LIN {X 0,Y 516.86,Z 224.104,A -85,B 0,C 180,E1 -4913.251,E2 -4913.251} C_VEL
LIN {X 0,Y 516.891,Z 224.097,A -85,B 0,C 180,E1 -4916.118,E2 -4916.118} C_VEL
LIN {X 0,Y 516.796,Z 224.113,A -85,B 0,C 180,E1 -4918.954,E2 -4918.954} C_VEL
LIN {X 0,Y 516.6,Z 224.138,A -85,B 0,C 180,E1 -4920.674,E2 -4920.674} C_VEL
LIN {X 0,Y 516.555,Z 225.784,A -85,B 0,C 180,E1 -4922.445,E2 -4922.445} C_VEL
LIN {X 0,Y 516.513,Z 229.358,A -85,B 0,C 180,E1 -4925.734,E2 -4925.734} C_VEL
LIN {X 0,Y 516.417,Z 232.326,A -85,B 0,C 180,E1 -4928.441,E2 -4928.441} C_VEL
LIN {X 0,Y 516.398,Z 235.073,A -85,B 0,C 180,E1 -4930.934,E2 -4930.934} C_VEL
LIN {X 0,Y 516.39,Z 237.798,A -85,B 0,C 180,E1 -4933.392,E2 -4933.392} C_VEL
LIN {X 0,Y 516.408,Z 240.566,A -85,B 0,C 180,E1 -4935.819,E2 -4935.819} C_VEL
LIN {X 0,Y 516.373,Z 244.264,A -85,B 0,C 180,E1 -4939.014,E2 -4939.014} C_VEL
LIN {X 0,Y 516.358,Z 245.702,A -85,B 0,C 180,E1 -4940.203,E2 -4940.203} C_VEL
LIN {X 0,Y 518.519,Z 256.334,A -85,B 0,C 180,E1 -4940.54,E2 -4940.54} C_VEL
LIN {X 0,Y 518.318,Z 269.35,A -85,B 0,C 180,E1 -4941.028,E2 -4941.028} C_VEL
LIN {X 0,Y 518.116,Z 280.838,A -85,B 0,C 180,E1 -4941.614,E2 -4941.614} C_VEL
LIN {X 0,Y 517.752,Z 291.503,A -85,B 0,C 180,E1 -4942.307,E2 -4942.307} C_VEL
LIN {X 0,Y 517.502,Z 302.062,A -85,B 0,C 180,E1 -4943.174,E2 -4943.174} C_VEL
LIN {X 0,Y 517.212,Z 311.692,A -85,B 0,C 180,E1 -4944.15,E2 -4944.15} C_VEL
LIN {X 0,Y 516.934,Z 319.598,A -85,B 0,C 180,E1 -4945.124,E2 -4945.124} C_VEL
LIN {X 0,Y 516.716,Z 327.363,A -85,B 0,C 180,E1 -4946.295,E2 -4946.295} C_VEL
LIN {X 0,Y 516.565,Z 332.623,A -85,B 0,C 180,E1 -4947.27,E2 -4947.27} C_VEL
LIN {X 0,Y 516.325,Z 337.788,A -85,B 0,C 180,E1 -4948.439,E2 -4948.439} C_VEL
LIN {X 0,Y 516.372,Z 341.79,A -85,B 0,C 180,E1 -4949.609,E2 -4949.609} C_VEL
LIN {X 0,Y 516.205,Z 344.784,A -85,B 0,C 180,E1 -4950.779,E2 -4950.779} C_VEL
LIN {X 0,Y 516.205,Z 346.261,A -85,B 0,C 180,E1 -4951.559,E2 -4951.559} C_VEL
LIN {X 0,Y 516.352,Z 347.941,A -85,B 0,C 180,E1 -4953.12,E2 -4953.12} C_VEL
LIN {X 0,Y 516.323,Z 348.221,A -85,B 0,C 180,E1 -4953.901,E2 -4953.901} C_VEL
LIN {X 0,Y 516.234,Z 348.118,A -85,B 0,C 180,E1 -4954.684,E2 -4954.684} C_VEL
LIN {X 0,Y 516.3,Z 347.579,A -85,B 0,C 180,E1 -4955.467,E2 -4955.467} C_VEL
LIN {X 0,Y 516.323,Z 345.343,A -85,B 0,C 180,E1 -4957.035,E2 -4957.035} C_VEL
LIN {X 0,Y 516.361,Z 342.554,A -85,B 0,C 180,E1 -4958.215,E2 -4958.215} C_VEL
LIN {X 0,Y 516.401,Z 338.739,A -85,B 0,C 180,E1 -4959.398,E2 -4959.398} C_VEL
LIN {X 0,Y 516.519,Z 333.78,A -85,B 0,C 180,E1 -4960.583,E2 -4960.583} C_VEL
LIN {X 0,Y 516.739,Z 327.523,A -85,B 0,C 180,E1 -4961.77,E2 -4961.77} C_VEL
LIN {X 0,Y 516.954,Z 319.645,A -85,B 0,C 180,E1 -4962.961,E2 -4962.961} C_VEL
LIN {X 0,Y 517.176,Z 311.578,A -85,B 0,C 180,E1 -4963.957,E2 -4963.957} C_VEL
LIN {X 0,Y 517.498,Z 301.699,A -85,B 0,C 180,E1 -4964.952,E2 -4964.952} C_VEL
LIN {X 0,Y 517.737,Z 291.95,A -85,B 0,C 180,E1 -4965.752,E2 -4965.752} C_VEL
LIN {X 0,Y 518.044,Z 281.356,A -85,B 0,C 180,E1 -4966.45,E2 -4966.45} C_VEL
LIN {X 0,Y 518.269,Z 268.518,A -85,B 0,C 180,E1 -4967.102,E2 -4967.102} C_VEL
LIN {X 0,Y 518.449,Z 255.755,A -85,B 0,C 180,E1 -4967.572,E2 -4967.572} C_VEL
LIN {X 0,Y 516.346,Z 245.639,A -85,B 0,C 180,E1 -4967.9,E2 -4967.9} C_VEL
LIN {X 0,Y 516.311,Z 242.393,A -85,B 0,C 180,E1 -4970.725,E2 -4970.725} C_VEL
LIN {X 0,Y 516.385,Z 239.494,A -85,B 0,C 180,E1 -4973.245,E2 -4973.245} C_VEL
LIN {X 0,Y 516.46,Z 236.317,A -85,B 0,C 180,E1 -4976.086,E2 -4976.086} C_VEL
LIN {X 0,Y 516.466,Z 233.733,A -85,B 0,C 180,E1 -4978.441,E2 -4978.441} C_VEL
LIN {X 0,Y 516.508,Z 230.848,A -85,B 0,C 180,E1 -4981.133,E2 -4981.133} C_VEL
LIN {X 0,Y 516.564,Z 227.881,A -85,B 0,C 180,E1 -4983.909,E2 -4983.909} C_VEL
LIN {X 0,Y 516.61,Z 224.866,A -85,B 0,C 180,E1 -4986.767,E2 -4986.767} C_VEL
LIN {X 0,Y 516.683,Z 224.128,A -85,B 0,C 180,E1 -4987.914,E2 -4987.914} C_VEL
LIN {X 0,Y 516.873,Z 224.101,A -85,B 0,C 180,E1 -4990.741,E2 -4990.741} C_VEL
LIN {X 0,Y 516.879,Z 224.103,A -85,B 0,C 180,E1 -4992.83,E2 -4992.83} C_VEL
LIN {X 0,Y 516.917,Z 224.094,A -85,B 0,C 180,E1 -4995.009,E2 -4995.009} C_VEL
LIN {X 0,Y 516.901,Z 224.096,A -85,B 0,C 180,E1 -4998.398,E2 -4998.398} C_VEL
LIN {X 0,Y 516.874,Z 224.101,A -85,B 0,C 180,E1 -5001.283,E2 -5001.283} C_VEL
LIN {X 0,Y 516.883,Z 224.103,A -85,B 0,C 180,E1 -5004.22,E2 -5004.22} C_VEL
LIN {X 0,Y 516.872,Z 224.1,A -85,B 0,C 180,E1 -5007.051,E2 -5007.051} C_VEL
LIN {X 0,Y 516.877,Z 224.099,A -85,B 0,C 180,E1 -5009.795,E2 -5009.795} C_VEL
LIN {X 0,Y 516.921,Z 224.097,A -85,B 0,C 180,E1 -5012.467,E2 -5012.467} C_VEL
LIN {X 0,Y 516.902,Z 224.095,A -85,B 0,C 180,E1 -5015.071,E2 -5015.071} C_VEL
LIN {X 0,Y 516.874,Z 224.099,A -85,B 0,C 180,E1 -5018.462,E2 -5018.462} C_VEL
LIN {X 0,Y 516.89,Z 224.1,A -85,B 0,C 180,E1 -5020.954,E2 -5020.954} C_VEL
LIN {X 0,Y 516.904,Z 224.096,A -85,B 0,C 180,E1 -5023.41,E2 -5023.41} C_VEL
LIN {X 0,Y 516.885,Z 224.101,A -85,B 0,C 180,E1 -5025.833,E2 -5025.833} C_VEL
LIN {X 0,Y 516.954,Z 224.089,A -85,B 0,C 180,E1 -5028.233,E2 -5028.233} C_VEL
LIN {X 0,Y 516.953,Z 224.089,A -85,B 0,C 180,E1 -5031.399,E2 -5031.399} C_VEL
LIN {X 0,Y 517.056,Z 224.077,A -85,B 0,C 180,E1 -5034.54,E2 -5034.54} C_VEL
LIN {X 0,Y 517.07,Z 224.075,A -85,B 0,C 180,E1 -5037.663,E2 -5037.663} C_VEL
LIN {X 0,Y 517.079,Z 224.076,A -85,B 0,C 180,E1 -5040.779,E2 -5040.779} C_VEL
LIN {X 0,Y 517.003,Z 224.083,A -85,B 0,C 180,E1 -5043.117,E2 -5043.117} C_VEL
LIN {X 0,Y 517.001,Z 224.083,A -85,B 0,C 180,E1 -5046.243,E2 -5046.243} C_VEL
LIN {X 0,Y 516.939,Z 224.091,A -85,B 0,C 180,E1 -5049.389,E2 -5049.389} C_VEL
LIN {X 0,Y 516.939,Z 224.094,A -85,B 0,C 180,E1 -5051.807,E2 -5051.807} C_VEL
LIN {X 0,Y 516.933,Z 224.095,A -85,B 0,C 180,E1 -5055.147,E2 -5055.147} C_VEL
LIN {X 0,Y 516.915,Z 224.095,A -85,B 0,C 180,E1 -5058.223,E2 -5058.223} C_VEL
LIN {X 0,Y 516.901,Z 224.097,A -85,B 0,C 180,E1 -5060.702,E2 -5060.702} C_VEL
LIN {X 0,Y 516.879,Z 224.099,A -85,B 0,C 180,E1 -5064.074,E2 -5064.074} C_VEL
LIN {X 0,Y 516.92,Z 224.097,A -85,B 0,C 180,E1 -5066.658,E2 -5066.658} C_VEL
LIN {X 0,Y 516.915,Z 224.094,A -85,B 0,C 180,E1 -5069.527,E2 -5069.527} C_VEL
LIN {X 0,Y 516.885,Z 224.098,A -85,B 0,C 180,E1 -5072.544,E2 -5072.544} C_VEL
LIN {X 0,Y 516.857,Z 224.104,A -85,B 0,C 180,E1 -5075.331,E2 -5075.331} C_VEL
LIN {X 0,Y 516.873,Z 224.1,A -85,B 0,C 180,E1 -5077.944,E2 -5077.944} C_VEL
LIN {X 0,Y 516.874,Z 224.099,A -85,B 0,C 180,E1 -5080.743,E2 -5080.743} C_VEL
LIN {X 0,Y 516.873,Z 224.1,A -85,B 0,C 180,E1 -5083.904,E2 -5083.904} C_VEL
LIN {X 0,Y 516.875,Z 224.102,A -85,B 0,C 180,E1 -5086.108,E2 -5086.108} C_VEL
LIN {X 0,Y 516.898,Z 224.1,A -85,B 0,C 180,E1 -5089.262,E2 -5089.262} C_VEL
LIN {X 0,Y 516.894,Z 224.132,A -85,B 0,C 180,E1 -5091.287,E2 -5091.287} C_VEL
LIN {X 0,Y 518.012,Z 230.689,A -85,B 0,C 180,E1 -5093.832,E2 -5093.832} C_VEL
LIN {X 0,Y 518.059,Z 236.321,A -85,B 0,C 180,E1 -5095.846,E2 -5095.846} C_VEL
LIN {X 0,Y 517.804,Z 244.803,A -85,B 0,C 180,E1 -5098.769,E2 -5098.769} C_VEL
LIN {X 0,Y 517.573,Z 254.623,A -85,B 0,C 180,E1 -5101.96,E2 -5101.96} C_VEL
LIN {X 0,Y 517.325,Z 262.962,A -85,B 0,C 180,E1 -5104.665,E2 -5104.665} C_VEL
LIN {X 0,Y 517.112,Z 272.229,A -85,B 0,C 180,E1 -5107.634,E2 -5107.634} C_VEL
LIN {X 0,Y 516.902,Z 281.496,A -85,B 0,C 180,E1 -5110.544,E2 -5110.544} C_VEL
LIN {X 0,Y 516.708,Z 290.764,A -85,B 0,C 180,E1 -5113.405,E2 -5113.405} C_VEL
LIN {X 0,Y 516.568,Z 299.534,A -85,B 0,C 180,E1 -5116.077,E2 -5116.077} C_VEL
LIN {X 0,Y 518.521,Z 312.228,A -85,B 0,C 180,E1 -5116.43,E2 -5116.43} C_VEL
LIN {X 0,Y 518.305,Z 323.804,A -85,B 0,C 180,E1 -5116.824,E2 -5116.824} C_VEL
LIN {X 0,Y 518,Z 335.432,A -85,B 0,C 180,E1 -5117.364,E2 -5117.364} C_VEL
LIN {X 0,Y 517.656,Z 347.73,A -85,B 0,C 180,E1 -5118.119,E2 -5118.119} C_VEL
LIN {X 0,Y 517.41,Z 358.276,A -85,B 0,C 180,E1 -5118.94,E2 -5118.94} C_VEL
LIN {X 0,Y 517.093,Z 367.551,A -85,B 0,C 180,E1 -5119.824,E2 -5119.824} C_VEL
LIN {X 0,Y 516.866,Z 376,A -85,B 0,C 180,E1 -5120.808,E2 -5120.808} C_VEL
LIN {X 0,Y 516.639,Z 384.244,A -85,B 0,C 180,E1 -5121.986,E2 -5121.986} C_VEL
LIN {X 0,Y 516.478,Z 391.083,A -85,B 0,C 180,E1 -5123.202,E2 -5123.202} C_VEL
LIN {X 0,Y 516.405,Z 396.954,A -85,B 0,C 180,E1 -5124.535,E2 -5124.535} C_VEL
LIN {X 0,Y 516.343,Z 400.898,A -85,B 0,C 180,E1 -5125.708,E2 -5125.708} C_VEL
LIN {X 0,Y 516.282,Z 403.81,A -85,B 0,C 180,E1 -5126.88,E2 -5126.88} C_VEL
LIN {X 0,Y 516.261,Z 405.198,A -85,B 0,C 180,E1 -5127.661,E2 -5127.661} C_VEL
LIN {X 0,Y 516.16,Z 406.786,A -85,B 0,C 180,E1 -5129.221,E2 -5129.221} C_VEL
LIN {X 0,Y 516.154,Z 407,A -85,B 0,C 180,E1 -5130.001,E2 -5130.001} C_VEL
LIN {X 0,Y 516.192,Z 406.184,A -85,B 0,C 180,E1 -5131.562,E2 -5131.562} C_VEL
LIN {X 0,Y 516.261,Z 405.197,A -85,B 0,C 180,E1 -5132.342,E2 -5132.342} C_VEL
LIN {X 0,Y 516.283,Z 403.808,A -85,B 0,C 180,E1 -5133.122,E2 -5133.122} C_VEL
LIN {X 0,Y 516.344,Z 400.892,A -85,B 0,C 180,E1 -5134.294,E2 -5134.294} C_VEL
LIN {X 0,Y 516.406,Z 396.945,A -85,B 0,C 180,E1 -5135.468,E2 -5135.468} C_VEL
LIN {X 0,Y 516.488,Z 391.026,A -85,B 0,C 180,E1 -5136.809,E2 -5136.809} C_VEL
LIN {X 0,Y 516.642,Z 384.23,A -85,B 0,C 180,E1 -5138.016,E2 -5138.016} C_VEL
LIN {X 0,Y 516.868,Z 375.983,A -85,B 0,C 180,E1 -5139.195,E2 -5139.195} C_VEL
LIN {X 0,Y 517.094,Z 367.528,A -85,B 0,C 180,E1 -5140.178,E2 -5140.178} C_VEL
LIN {X 0,Y 517.454,Z 357.083,A -85,B 0,C 180,E1 -5141.161,E2 -5141.161} C_VEL
LIN {X 0,Y 517.707,Z 345.717,A -85,B 0,C 180,E1 -5142.02,E2 -5142.02} C_VEL
LIN {X 0,Y 517.984,Z 335.389,A -85,B 0,C 180,E1 -5142.639,E2 -5142.639} C_VEL
LIN {X 0,Y 518.256,Z 323.735,A -85,B 0,C 180,E1 -5143.18,E2 -5143.18} C_VEL
LIN {X 0,Y 518.415,Z 310.764,A -85,B 0,C 180,E1 -5143.612,E2 -5143.612} C_VEL
LIN {X 0,Y 516.567,Z 299.527,A -85,B 0,C 180,E1 -5143.926,E2 -5143.926} C_VEL
LIN {X 0,Y 516.712,Z 290.756,A -85,B 0,C 180,E1 -5146.598,E2 -5146.598} C_VEL
LIN {X 0,Y 516.908,Z 281.489,A -85,B 0,C 180,E1 -5149.459,E2 -5149.459} C_VEL
LIN {X 0,Y 517.102,Z 271.96,A -85,B 0,C 180,E1 -5152.452,E2 -5152.452} C_VEL
LIN {X 0,Y 517.324,Z 262.954,A -85,B 0,C 180,E1 -5155.338,E2 -5155.338} C_VEL
LIN {X 0,Y 517.606,Z 253.624,A -85,B 0,C 180,E1 -5158.375,E2 -5158.375} C_VEL
LIN {X 0,Y 517.852,Z 243.91,A -85,B 0,C 180,E1 -5161.552,E2 -5161.552} C_VEL
LIN {X 0,Y 518.058,Z 236.324,A -85,B 0,C 180,E1 -5164.154,E2 -5164.154} C_VEL
LIN {X 0,Y 518.027,Z 230.704,A -85,B 0,C 180,E1 -5166.169,E2 -5166.169} C_VEL
LIN {X 0,Y 516.895,Z 224.102,A -85,B 0,C 180,E1 -5168.775,E2 -5168.775} C_VEL
LIN {X 0,Y 516.913,Z 224.098,A -85,B 0,C 180,E1 -5171.776,E2 -5171.776} C_VEL
LIN {X 0,Y 516.93,Z 224.094,A -85,B 0,C 180,E1 -5175.011,E2 -5175.011} C_VEL
LIN {X 0,Y 516.92,Z 224.094,A -85,B 0,C 180,E1 -5178.399,E2 -5178.399} C_VEL
LIN {X 0,Y 516.883,Z 224.101,A -85,B 0,C 180,E1 -5181.284,E2 -5181.284} C_VEL
LIN {X 0,Y 516.862,Z 224.101,A -85,B 0,C 180,E1 -5184.219,E2 -5184.219} C_VEL
LIN {X 0,Y 516.873,Z 224.099,A -85,B 0,C 180,E1 -5187.051,E2 -5187.051} C_VEL
LIN {X 0,Y 516.887,Z 224.1,A -85,B 0,C 180,E1 -5189.796,E2 -5189.796} C_VEL
LIN {X 0,Y 516.904,Z 224.096,A -85,B 0,C 180,E1 -5192.466,E2 -5192.466} C_VEL
LIN {X 0,Y 516.874,Z 224.103,A -85,B 0,C 180,E1 -5195.07,E2 -5195.07} C_VEL
LIN {X 0,Y 516.876,Z 224.1,A -85,B 0,C 180,E1 -5197.622,E2 -5197.622} C_VEL
LIN {X 0,Y 516.936,Z 224.093,A -85,B 0,C 180,E1 -5200.13,E2 -5200.13} C_VEL
LIN {X 0,Y 516.885,Z 224.1,A -85,B 0,C 180,E1 -5202.595,E2 -5202.595} C_VEL
LIN {X 0,Y 516.937,Z 224.09,A -85,B 0,C 180,E1 -5205.03,E2 -5205.03} C_VEL
LIN {X 0,Y 516.932,Z 224.092,A -85,B 0,C 180,E1 -5208.233,E2 -5208.233} C_VEL
LIN {X 0,Y 516.953,Z 224.095,A -85,B 0,C 180,E1 -5211.399,E2 -5211.399} C_VEL
LIN {X 0,Y 517.007,Z 224.083,A -85,B 0,C 180,E1 -5213.757,E2 -5213.757} C_VEL
LIN {X 0,Y 517.017,Z 224.085,A -85,B 0,C 180,E1 -5216.883,E2 -5216.883} C_VEL
LIN {X 0,Y 517.093,Z 224.077,A -85,B 0,C 180,E1 -5220,E2 -5220} C_VEL
LIN {X 0,Y 517.084,Z 224.074,A -85,B 0,C 180,E1 -5222.337,E2 -5222.337} C_VEL
LIN {X 0,Y 516.984,Z 224.091,A -85,B 0,C 180,E1 -5225.461,E2 -5225.461} C_VEL
LIN {X 0,Y 516.934,Z 224.092,A -85,B 0,C 180,E1 -5228.601,E2 -5228.601} C_VEL
LIN {X 0,Y 516.96,Z 224.088,A -85,B 0,C 180,E1 -5231.807,E2 -5231.807} C_VEL
LIN {X 0,Y 516.953,Z 224.09,A -85,B 0,C 180,E1 -5235.146,E2 -5235.146} C_VEL
LIN {X 0,Y 516.924,Z 224.096,A -85,B 0,C 180,E1 -5238.222,E2 -5238.222} C_VEL
LIN {X 0,Y 516.912,Z 224.095,A -85,B 0,C 180,E1 -5240.702,E2 -5240.702} C_VEL
LIN {X 0,Y 516.862,Z 224.105,A -85,B 0,C 180,E1 -5243.224,E2 -5243.224} C_VEL
LIN {X 0,Y 516.862,Z 224.1,A -85,B 0,C 180,E1 -5246.176,E2 -5246.176} C_VEL
LIN {X 0,Y 516.91,Z 224.094,A -85,B 0,C 180,E1 -5249.305,E2 -5249.305} C_VEL
LIN {X 0,Y 516.902,Z 224.097,A -85,B 0,C 180,E1 -5252.543,E2 -5252.543} C_VEL
LIN {X 0,Y 516.871,Z 224.103,A -85,B 0,C 180,E1 -5255.329,E2 -5255.329} C_VEL
LIN {X 0,Y 516.886,Z 224.099,A -85,B 0,C 180,E1 -5257.942,E2 -5257.942} C_VEL
LIN {X 0,Y 516.879,Z 224.103,A -85,B 0,C 180,E1 -5260.743,E2 -5260.743} C_VEL
LIN {X 0,Y 516.888,Z 224.098,A -85,B 0,C 180,E1 -5263.903,E2 -5263.903} C_VEL
LIN {X 0,Y 516.831,Z 224.102,A -85,B 0,C 180,E1 -5266.861,E2 -5266.861} C_VEL
LIN {X 0,Y 516.839,Z 224.106,A -85,B 0,C 180,E1 -5269.596,E2 -5269.596} C_VEL
LIN {X 0,Y 516.852,Z 224.103,A -85,B 0,C 180,E1 -5270.247,E2 -5270.247} C_VEL
LIN {X 0,Y 516.226,Z 224.184,A -85,B 0,C 180,E1 -5270.898,E2 -5270.898} C_VEL
LIN {X 0,Y 513.387,Z 224.543,A -85,B 0,C 180,E1 -5271.953,E2 -5271.953} C_VEL
LIN {X 0,Y 510.958,Z 224.846,A -85,B 0,C 180,E1 -5272.804,E2 -5272.804} C_VEL
LIN {X 0,Y 509.905,Z 224.973,A -85,B 0,C 180,E1 -5273.46,E2 -5273.46} C_VEL
LIN {X 0,Y 509.815,Z 224.982,A -85,B 0,C 180,E1 -5273.683,E2 -5273.683} C_VEL
LIN {X 0,Y 509.844,Z 224.978,A -85,B 0,C 180,E1 -5276.537,E2 -5276.537} C_VEL
LIN {X 0,Y 509.702,Z 224.998,A -85,B 0,C 180,E1 -5279.324,E2 -5279.324} C_VEL
LIN {X 0,Y 509.493,Z 225.07,A -85,B 0,C 180,E1 -5281.131,E2 -5281.131} C_VEL
LIN {X 0,Y 509.441,Z 227.945,A -85,B 0,C 180,E1 -5283.802,E2 -5283.802} C_VEL
LIN {X 0,Y 509.415,Z 230.768,A -85,B 0,C 180,E1 -5286.415,E2 -5286.415} C_VEL
LIN {X 0,Y 509.381,Z 234.482,A -85,B 0,C 180,E1 -5289.821,E2 -5289.821} C_VEL
LIN {X 0,Y 509.386,Z 237.231,A -85,B 0,C 180,E1 -5292.329,E2 -5292.329} C_VEL
LIN {X 0,Y 509.341,Z 240.937,A -85,B 0,C 180,E1 -5295.618,E2 -5295.618} C_VEL
LIN {X 0,Y 509.323,Z 244.681,A -85,B 0,C 180,E1 -5298.86,E2 -5298.86} C_VEL
LIN {X 0,Y 509.269,Z 246.038,A -85,B 0,C 180,E1 -5299.99,E2 -5299.99} C_VEL
LIN {X 0,Y 511.67,Z 257.697,A -85,B 0,C 180,E1 -5300.387,E2 -5300.387} C_VEL
LIN {X 0,Y 511.407,Z 271.035,A -85,B 0,C 180,E1 -5300.906,E2 -5300.906} C_VEL
LIN {X 0,Y 511.178,Z 282.233,A -85,B 0,C 180,E1 -5301.5,E2 -5301.5} C_VEL
LIN {X 0,Y 510.79,Z 292.637,A -85,B 0,C 180,E1 -5302.2,E2 -5302.2} C_VEL
LIN {X 0,Y 510.54,Z 303.081,A -85,B 0,C 180,E1 -5303.081,E2 -5303.081} C_VEL
LIN {X 0,Y 510.221,Z 312.613,A -85,B 0,C 180,E1 -5304.069,E2 -5304.069} C_VEL
LIN {X 0,Y 509.916,Z 320.438,A -85,B 0,C 180,E1 -5305.057,E2 -5305.057} C_VEL
LIN {X 0,Y 509.683,Z 328.108,A -85,B 0,C 180,E1 -5306.243,E2 -5306.243} C_VEL
LIN {X 0,Y 509.325,Z 335.152,A -85,B 0,C 180,E1 -5307.626,E2 -5307.626} C_VEL
LIN {X 0,Y 509.351,Z 339.841,A -85,B 0,C 180,E1 -5308.813,E2 -5308.813} C_VEL
LIN {X 0,Y 509.166,Z 343.465,A -85,B 0,C 180,E1 -5309.999,E2 -5309.999} C_VEL
LIN {X 0,Y 509.123,Z 345.335,A -85,B 0,C 180,E1 -5310.79,E2 -5310.79} C_VEL
LIN {X 0,Y 509.125,Z 346.768,A -85,B 0,C 180,E1 -5311.581,E2 -5311.581} C_VEL
LIN {X 0,Y 509.275,Z 348.401,A -85,B 0,C 180,E1 -5313.163,E2 -5313.163} C_VEL
LIN {X 0,Y 509.249,Z 348.658,A -85,B 0,C 180,E1 -5313.956,E2 -5313.956} C_VEL
LIN {X 0,Y 509.15,Z 348.516,A -85,B 0,C 180,E1 -5314.749,E2 -5314.749} C_VEL
LIN {X 0,Y 509.231,Z 347.949,A -85,B 0,C 180,E1 -5315.543,E2 -5315.543} C_VEL
LIN {X 0,Y 509.262,Z 345.668,A -85,B 0,C 180,E1 -5317.134,E2 -5317.134} C_VEL
LIN {X 0,Y 509.297,Z 342.832,A -85,B 0,C 180,E1 -5318.33,E2 -5318.33} C_VEL
LIN {X 0,Y 509.341,Z 338.966,A -85,B 0,C 180,E1 -5319.53,E2 -5319.53} C_VEL
LIN {X 0,Y 509.484,Z 333.952,A -85,B 0,C 180,E1 -5320.731,E2 -5320.731} C_VEL
LIN {X 0,Y 509.71,Z 327.615,A -85,B 0,C 180,E1 -5321.935,E2 -5321.935} C_VEL
LIN {X 0,Y 509.95,Z 319.65,A -85,B 0,C 180,E1 -5323.143,E2 -5323.143} C_VEL
LIN {X 0,Y 510.194,Z 311.498,A -85,B 0,C 180,E1 -5324.152,E2 -5324.152} C_VEL
LIN {X 0,Y 510.561,Z 301.516,A -85,B 0,C 180,E1 -5325.16,E2 -5325.16} C_VEL
LIN {X 0,Y 510.823,Z 291.602,A -85,B 0,C 180,E1 -5325.97,E2 -5325.97} C_VEL
LIN {X 0,Y 511.171,Z 280.773,A -85,B 0,C 180,E1 -5326.678,E2 -5326.678} C_VEL
LIN {X 0,Y 511.381,Z 268.79,A -85,B 0,C 180,E1 -5327.288,E2 -5327.288} C_VEL
LIN {X 0,Y 511.547,Z 256.515,A -85,B 0,C 180,E1 -5327.747,E2 -5327.747} C_VEL
LIN {X 0,Y 509.267,Z 246.036,A -85,B 0,C 180,E1 -5328.095,E2 -5328.095} C_VEL
LIN {X 0,Y 509.233,Z 242.651,A -85,B 0,C 180,E1 -5331.027,E2 -5331.027} C_VEL
LIN {X 0,Y 509.298,Z 239.741,A -85,B 0,C 180,E1 -5333.588,E2 -5333.588} C_VEL
LIN {X 0,Y 509.403,Z 236.778,A -85,B 0,C 180,E1 -5336.262,E2 -5336.262} C_VEL
LIN {X 0,Y 509.417,Z 233.946,A -85,B 0,C 180,E1 -5338.871,E2 -5338.871} C_VEL
LIN {X 0,Y 509.419,Z 231.033,A -85,B 0,C 180,E1 -5341.616,E2 -5341.616} C_VEL
LIN {X 0,Y 509.517,Z 228.043,A -85,B 0,C 180,E1 -5344.438,E2 -5344.438} C_VEL
LIN {X 0,Y 509.545,Z 225.018,A -85,B 0,C 180,E1 -5347.362,E2 -5347.362} C_VEL
LIN {X 0,Y 509.762,Z 224.99,A -85,B 0,C 180,E1 -5349.46,E2 -5349.46} C_VEL
LIN {X 0,Y 509.853,Z 224.974,A -85,B 0,C 180,E1 -5351.896,E2 -5351.896} C_VEL
LIN {X 0,Y 509.85,Z 224.975,A -85,B 0,C 180,E1 -5355.331,E2 -5355.331} C_VEL
LIN {X 0,Y 509.843,Z 224.975,A -85,B 0,C 180,E1 -5358.573,E2 -5358.573} C_VEL
LIN {X 0,Y 509.843,Z 224.975,A -85,B 0,C 180,E1 -5361.785,E2 -5361.785} C_VEL
LIN {X 0,Y 509.838,Z 224.977,A -85,B 0,C 180,E1 -5364.622,E2 -5364.622} C_VEL
LIN {X 0,Y 509.85,Z 224.979,A -85,B 0,C 180,E1 -5367.48,E2 -5367.48} C_VEL
LIN {X 0,Y 509.848,Z 224.974,A -85,B 0,C 180,E1 -5370.273,E2 -5370.273} C_VEL
LIN {X 0,Y 509.878,Z 224.971,A -85,B 0,C 180,E1 -5372.944,E2 -5372.944} C_VEL
LIN {X 0,Y 509.861,Z 224.976,A -85,B 0,C 180,E1 -5375.573,E2 -5375.573} C_VEL
LIN {X 0,Y 509.839,Z 224.981,A -85,B 0,C 180,E1 -5378.998,E2 -5378.998} C_VEL
LIN {X 0,Y 509.87,Z 224.973,A -85,B 0,C 180,E1 -5382.001,E2 -5382.001} C_VEL
LIN {X 0,Y 509.899,Z 224.968,A -85,B 0,C 180,E1 -5384.818,E2 -5384.818} C_VEL
LIN {X 0,Y 509.89,Z 224.969,A -85,B 0,C 180,E1 -5388.123,E2 -5388.123} C_VEL
LIN {X 0,Y 509.898,Z 224.968,A -85,B 0,C 180,E1 -5391.279,E2 -5391.279} C_VEL
LIN {X 0,Y 509.974,Z 224.962,A -85,B 0,C 180,E1 -5393.67,E2 -5393.67} C_VEL
LIN {X 0,Y 509.949,Z 224.964,A -85,B 0,C 180,E1 -5396.84,E2 -5396.84} C_VEL
LIN {X 0,Y 510.05,Z 224.951,A -85,B 0,C 180,E1 -5399.21,E2 -5399.21} C_VEL
LIN {X 0,Y 510.043,Z 224.953,A -85,B 0,C 180,E1 -5402.369,E2 -5402.369} C_VEL
LIN {X 0,Y 509.997,Z 224.96,A -85,B 0,C 180,E1 -5405.535,E2 -5405.535} C_VEL
LIN {X 0,Y 509.94,Z 224.963,A -85,B 0,C 180,E1 -5407.922,E2 -5407.922} C_VEL
LIN {X 0,Y 509.899,Z 224.967,A -85,B 0,C 180,E1 -5411.126,E2 -5411.126} C_VEL
LIN {X 0,Y 509.851,Z 224.973,A -85,B 0,C 180,E1 -5414.366,E2 -5414.366} C_VEL
LIN {X 0,Y 509.892,Z 224.969,A -85,B 0,C 180,E1 -5417.652,E2 -5417.652} C_VEL
LIN {X 0,Y 509.875,Z 224.975,A -85,B 0,C 180,E1 -5420.402,E2 -5420.402} C_VEL
LIN {X 0,Y 509.81,Z 224.985,A -85,B 0,C 180,E1 -5423.564,E2 -5423.564} C_VEL
LIN {X 0,Y 509.904,Z 224.968,A -85,B 0,C 180,E1 -5426.38,E2 -5426.38} C_VEL
LIN {X 0,Y 509.876,Z 224.973,A -85,B 0,C 180,E1 -5428.844,E2 -5428.844} C_VEL
LIN {X 0,Y 509.811,Z 224.983,A -85,B 0,C 180,E1 -5431.591,E2 -5431.591} C_VEL
LIN {X 0,Y 509.837,Z 224.976,A -85,B 0,C 180,E1 -5434.415,E2 -5434.415} C_VEL
LIN {X 0,Y 509.808,Z 224.979,A -85,B 0,C 180,E1 -5437.342,E2 -5437.342} C_VEL
LIN {X 0,Y 509.829,Z 224.979,A -85,B 0,C 180,E1 -5440.383,E2 -5440.383} C_VEL
LIN {X 0,Y 509.796,Z 224.984,A -85,B 0,C 180,E1 -5443.061,E2 -5443.061} C_VEL
LIN {X 0,Y 509.823,Z 224.979,A -85,B 0,C 180,E1 -5445.793,E2 -5445.793} C_VEL
LIN {X 0,Y 509.86,Z 224.978,A -85,B 0,C 180,E1 -5448.577,E2 -5448.577} C_VEL
LIN {X 0,Y 509.856,Z 225.048,A -85,B 0,C 180,E1 -5451.032,E2 -5451.032} C_VEL
LIN {X 0,Y 511.037,Z 231.882,A -85,B 0,C 180,E1 -5453.749,E2 -5453.749} C_VEL
LIN {X 0,Y 511.085,Z 237.214,A -85,B 0,C 180,E1 -5455.683,E2 -5455.683} C_VEL
LIN {X 0,Y 510.844,Z 245.373,A -85,B 0,C 180,E1 -5458.537,E2 -5458.537} C_VEL
LIN {X 0,Y 510.579,Z 253.371,A -85,B 0,C 180,E1 -5461.201,E2 -5461.201} C_VEL
LIN {X 0,Y 510.385,Z 261.582,A -85,B 0,C 180,E1 -5463.857,E2 -5463.857} C_VEL
LIN {X 0,Y 510.121,Z 270.905,A -85,B 0,C 180,E1 -5466.882,E2 -5466.882} C_VEL
LIN {X 0,Y 509.92,Z 280.173,A -85,B 0,C 180,E1 -5469.846,E2 -5469.846} C_VEL
LIN {X 0,Y 509.714,Z 289.44,A -85,B 0,C 180,E1 -5472.757,E2 -5472.757} C_VEL
LIN {X 0,Y 509.527,Z 299.534,A -85,B 0,C 180,E1 -5475.881,E2 -5475.881} C_VEL
LIN {X 0,Y 511.612,Z 313.141,A -85,B 0,C 180,E1 -5476.269,E2 -5476.269} C_VEL
LIN {X 0,Y 511.371,Z 325.012,A -85,B 0,C 180,E1 -5476.692,E2 -5476.692} C_VEL
LIN {X 0,Y 511.018,Z 337.196,A -85,B 0,C 180,E1 -5477.289,E2 -5477.289} C_VEL
LIN {X 0,Y 510.69,Z 348.101,A -85,B 0,C 180,E1 -5477.981,E2 -5477.981} C_VEL
LIN {X 0,Y 510.37,Z 359.414,A -85,B 0,C 180,E1 -5478.886,E2 -5478.886} C_VEL
LIN {X 0,Y 510.034,Z 369.345,A -85,B 0,C 180,E1 -5479.883,E2 -5479.883} C_VEL
LIN {X 0,Y 509.759,Z 378.969,A -85,B 0,C 180,E1 -5481.078,E2 -5481.078} C_VEL
LIN {X 0,Y 509.52,Z 386.628,A -85,B 0,C 180,E1 -5482.272,E2 -5482.272} C_VEL
LIN {X 0,Y 509.335,Z 393.685,A -85,B 0,C 180,E1 -5483.664,E2 -5483.664} C_VEL
LIN {X 0,Y 509.247,Z 398.377,A -85,B 0,C 180,E1 -5484.855,E2 -5484.855} C_VEL
LIN {X 0,Y 509.253,Z 401.961,A -85,B 0,C 180,E1 -5486.044,E2 -5486.044} C_VEL
LIN {X 0,Y 509.2,Z 403.81,A -85,B 0,C 180,E1 -5486.836,E2 -5486.836} C_VEL
LIN {X 0,Y 509.161,Z 405.197,A -85,B 0,C 180,E1 -5487.628,E2 -5487.628} C_VEL
LIN {X 0,Y 509.073,Z 406.786,A -85,B 0,C 180,E1 -5489.21,E2 -5489.21} C_VEL
LIN {X 0,Y 509.065,Z 407,A -85,B 0,C 180,E1 -5490.001,E2 -5490.001} C_VEL
LIN {X 0,Y 509.113,Z 406.184,A -85,B 0,C 180,E1 -5491.583,E2 -5491.583} C_VEL
LIN {X 0,Y 509.161,Z 405.196,A -85,B 0,C 180,E1 -5492.374,E2 -5492.374} C_VEL
LIN {X 0,Y 509.201,Z 403.808,A -85,B 0,C 180,E1 -5493.166,E2 -5493.166} C_VEL
LIN {X 0,Y 509.234,Z 400.892,A -85,B 0,C 180,E1 -5494.354,E2 -5494.354} C_VEL
LIN {X 0,Y 509.345,Z 396.944,A -85,B 0,C 180,E1 -5495.544,E2 -5495.544} C_VEL
LIN {X 0,Y 509.411,Z 391.276,A -85,B 0,C 180,E1 -5496.854,E2 -5496.854} C_VEL
LIN {X 0,Y 509.586,Z 384.23,A -85,B 0,C 180,E1 -5498.128,E2 -5498.128} C_VEL
LIN {X 0,Y 509.847,Z 375.983,A -85,B 0,C 180,E1 -5499.322,E2 -5499.322} C_VEL
LIN {X 0,Y 510.083,Z 367.529,A -85,B 0,C 180,E1 -5500.319,E2 -5500.319} C_VEL
LIN {X 0,Y 510.48,Z 357.082,A -85,B 0,C 180,E1 -5501.315,E2 -5501.315} C_VEL
LIN {X 0,Y 510.739,Z 346.459,A -85,B 0,C 180,E1 -5502.134,E2 -5502.134} C_VEL
LIN {X 0,Y 511.046,Z 335.388,A -85,B 0,C 180,E1 -5502.813,E2 -5502.813} C_VEL
LIN {X 0,Y 511.359,Z 323.735,A -85,B 0,C 180,E1 -5503.361,E2 -5503.361} C_VEL
LIN {X 0,Y 511.431,Z 311.221,A -85,B 0,C 180,E1 -5503.789,E2 -5503.789} C_VEL
LIN {X 0,Y 509.527,Z 299.527,A -85,B 0,C 180,E1 -5504.122,E2 -5504.122} C_VEL
LIN {X 0,Y 509.719,Z 289.432,A -85,B 0,C 180,E1 -5507.245,E2 -5507.245} C_VEL
LIN {X 0,Y 509.95,Z 279.332,A -85,B 0,C 180,E1 -5510.42,E2 -5510.42} C_VEL
LIN {X 0,Y 510.18,Z 269.574,A -85,B 0,C 180,E1 -5513.547,E2 -5513.547} C_VEL
LIN {X 0,Y 510.43,Z 260.485,A -85,B 0,C 180,E1 -5516.495,E2 -5516.495} C_VEL
LIN {X 0,Y 510.59,Z 252.049,A -85,B 0,C 180,E1 -5519.252,E2 -5519.252} C_VEL
LIN {X 0,Y 510.87,Z 243.847,A -85,B 0,C 180,E1 -5521.982,E2 -5521.982} C_VEL
LIN {X 0,Y 511.154,Z 235.883,A -85,B 0,C 180,E1 -5524.794,E2 -5524.794} C_VEL
LIN {X 0,Y 511.047,Z 231.896,A -85,B 0,C 180,E1 -5526.253,E2 -5526.253} C_VEL
LIN {X 0,Y 509.849,Z 224.979,A -85,B 0,C 180,E1 -5529.035,E2 -5529.035} C_VEL
LIN {X 0,Y 509.858,Z 224.978,A -85,B 0,C 180,E1 -5531.897,E2 -5531.897} C_VEL
LIN {X 0,Y 509.864,Z 224.976,A -85,B 0,C 180,E1 -5535.333,E2 -5535.333} C_VEL
LIN {X 0,Y 509.862,Z 224.973,A -85,B 0,C 180,E1 -5538.575,E2 -5538.575} C_VEL
LIN {X 0,Y 509.855,Z 224.973,A -85,B 0,C 180,E1 -5541.787,E2 -5541.787} C_VEL
LIN {X 0,Y 509.824,Z 224.983,A -85,B 0,C 180,E1 -5544.621,E2 -5544.621} C_VEL
LIN {X 0,Y 509.841,Z 224.974,A -85,B 0,C 180,E1 -5547.479,E2 -5547.479} C_VEL
LIN {X 0,Y 509.864,Z 224.976,A -85,B 0,C 180,E1 -5550.274,E2 -5550.274} C_VEL
LIN {X 0,Y 509.891,Z 224.973,A -85,B 0,C 180,E1 -5553.628,E2 -5553.628} C_VEL
LIN {X 0,Y 509.829,Z 224.978,A -85,B 0,C 180,E1 -5556.436,E2 -5556.436} C_VEL
LIN {X 0,Y 509.923,Z 224.965,A -85,B 0,C 180,E1 -5559.845,E2 -5559.845} C_VEL
LIN {X 0,Y 509.859,Z 224.978,A -85,B 0,C 180,E1 -5562.347,E2 -5562.347} C_VEL
LIN {X 0,Y 509.891,Z 224.968,A -85,B 0,C 180,E1 -5564.818,E2 -5564.818} C_VEL
LIN {X 0,Y 509.896,Z 224.97,A -85,B 0,C 180,E1 -5568.131,E2 -5568.131} C_VEL
LIN {X 0,Y 509.899,Z 224.972,A -85,B 0,C 180,E1 -5571.28,E2 -5571.28} C_VEL
LIN {X 0,Y 509.959,Z 224.962,A -85,B 0,C 180,E1 -5573.67,E2 -5573.67} C_VEL
LIN {X 0,Y 510.06,Z 224.949,A -85,B 0,C 180,E1 -5577.631,E2 -5577.631} C_VEL
LIN {X 0,Y 510.064,Z 224.952,A -85,B 0,C 180,E1 -5580,E2 -5580} C_VEL
LIN {X 0,Y 510.054,Z 224.95,A -85,B 0,C 180,E1 -5582.369,E2 -5582.369} C_VEL
LIN {X 0,Y 509.937,Z 224.968,A -85,B 0,C 180,E1 -5585.536,E2 -5585.536} C_VEL
LIN {X 0,Y 509.883,Z 224.969,A -85,B 0,C 180,E1 -5587.923,E2 -5587.923} C_VEL
LIN {X 0,Y 509.915,Z 224.969,A -85,B 0,C 180,E1 -5591.126,E2 -5591.126} C_VEL
LIN {X 0,Y 509.869,Z 224.975,A -85,B 0,C 180,E1 -5594.366,E2 -5594.366} C_VEL
LIN {X 0,Y 509.88,Z 224.971,A -85,B 0,C 180,E1 -5596.826,E2 -5596.826} C_VEL
LIN {X 0,Y 509.923,Z 224.967,A -85,B 0,C 180,E1 -5600.155,E2 -5600.155} C_VEL
LIN {X 0,Y 509.818,Z 224.98,A -85,B 0,C 180,E1 -5603.564,E2 -5603.564} C_VEL
LIN {X 0,Y 509.803,Z 224.981,A -85,B 0,C 180,E1 -5606.352,E2 -5606.352} C_VEL
LIN {X 0,Y 509.842,Z 224.977,A -85,B 0,C 180,E1 -5608.847,E2 -5608.847} C_VEL
LIN {X 0,Y 509.826,Z 224.978,A -85,B 0,C 180,E1 -5611.59,E2 -5611.59} C_VEL
LIN {X 0,Y 509.845,Z 224.976,A -85,B 0,C 180,E1 -5614.414,E2 -5614.414} C_VEL
LIN {X 0,Y 509.816,Z 224.982,A -85,B 0,C 180,E1 -5617.341,E2 -5617.341} C_VEL
LIN {X 0,Y 509.841,Z 224.976,A -85,B 0,C 180,E1 -5620.382,E2 -5620.382} C_VEL
LIN {X 0,Y 509.808,Z 224.981,A -85,B 0,C 180,E1 -5623.059,E2 -5623.059} C_VEL
LIN {X 0,Y 509.813,Z 224.979,A -85,B 0,C 180,E1 -5625.795,E2 -5625.795} C_VEL
LIN {X 0,Y 509.79,Z 224.981,A -85,B 0,C 180,E1 -5628.567,E2 -5628.567} C_VEL
LIN {X 0,Y 509.855,Z 224.978,A -85,B 0,C 180,E1 -5631.786,E2 -5631.786} C_VEL
LIN {X 0,Y 509.815,Z 224.982,A -85,B 0,C 180,E1 -5633.683,E2 -5633.683} C_VEL
LIN {X 0,Y 509.151,Z 225.062,A -85,B 0,C 180,E1 -5634.343,E2 -5634.343} C_VEL
LIN {X 0,Y 506.336,Z 225.416,A -85,B 0,C 180,E1 -5635.415,E2 -5635.415} C_VEL
LIN {X 0,Y 503.941,Z 225.716,A -85,B 0,C 180,E1 -5636.278,E2 -5636.278} C_VEL
LIN {X 0,Y 502.886,Z 225.845,A -85,B 0,C 180,E1 -5636.944,E2 -5636.944} C_VEL
LIN {X 0,Y 502.786,Z 225.856,A -85,B 0,C 180,E1 -5637.17,E2 -5637.17} C_VEL
LIN {X 0,Y 502.595,Z 225.883,A -85,B 0,C 180,E1 -5639.773,E2 -5639.773} C_VEL
LIN {X 0,Y 502.425,Z 226.289,A -85,B 0,C 180,E1 -5641.601,E2 -5641.601} C_VEL
LIN {X 0,Y 502.365,Z 229.168,A -85,B 0,C 180,E1 -5644.297,E2 -5644.297} C_VEL
LIN {X 0,Y 502.336,Z 232.009,A -85,B 0,C 180,E1 -5646.936,E2 -5646.936} C_VEL
LIN {X 0,Y 502.277,Z 235.745,A -85,B 0,C 180,E1 -5650.377,E2 -5650.377} C_VEL
LIN {X 0,Y 502.279,Z 238.51,A -85,B 0,C 180,E1 -5652.911,E2 -5652.911} C_VEL
LIN {X 0,Y 502.261,Z 241.322,A -85,B 0,C 180,E1 -5655.411,E2 -5655.411} C_VEL
LIN {X 0,Y 502.277,Z 245.104,A -85,B 0,C 180,E1 -5658.702,E2 -5658.702} C_VEL
LIN {X 0,Y 502.219,Z 246.399,A -85,B 0,C 180,E1 -5659.797,E2 -5659.797} C_VEL
LIN {X 0,Y 504.755,Z 258.335,A -85,B 0,C 180,E1 -5660.204,E2 -5660.204} C_VEL
LIN {X 0,Y 504.522,Z 271.607,A -85,B 0,C 180,E1 -5660.73,E2 -5660.73} C_VEL
LIN {X 0,Y 504.242,Z 283.553,A -85,B 0,C 180,E1 -5661.382,E2 -5661.382} C_VEL
LIN {X 0,Y 503.83,Z 293.764,A -85,B 0,C 180,E1 -5662.09,E2 -5662.09} C_VEL
LIN {X 0,Y 503.576,Z 304.101,A -85,B 0,C 180,E1 -5662.985,E2 -5662.985} C_VEL
LIN {X 0,Y 503.23,Z 313.535,A -85,B 0,C 180,E1 -5663.986,E2 -5663.986} C_VEL
LIN {X 0,Y 502.9,Z 321.277,A -85,B 0,C 180,E1 -5664.988,E2 -5664.988} C_VEL
LIN {X 0,Y 502.65,Z 328.845,A -85,B 0,C 180,E1 -5666.191,E2 -5666.191} C_VEL
LIN {X 0,Y 502.456,Z 334.031,A -85,B 0,C 180,E1 -5667.193,E2 -5667.193} C_VEL
LIN {X 0,Y 502.19,Z 339.074,A -85,B 0,C 180,E1 -5668.395,E2 -5668.395} C_VEL
LIN {X 0,Y 502.215,Z 342.979,A -85,B 0,C 180,E1 -5669.598,E2 -5669.598} C_VEL
LIN {X 0,Y 502.042,Z 345.885,A -85,B 0,C 180,E1 -5670.801,E2 -5670.801} C_VEL
LIN {X 0,Y 502.128,Z 348.255,A -85,B 0,C 180,E1 -5672.405,E2 -5672.405} C_VEL
LIN {X 0,Y 502.187,Z 348.861,A -85,B 0,C 180,E1 -5673.208,E2 -5673.208} C_VEL
LIN {X 0,Y 502.177,Z 349.094,A -85,B 0,C 180,E1 -5674.011,E2 -5674.011} C_VEL
LIN {X 0,Y 502.07,Z 348.909,A -85,B 0,C 180,E1 -5674.817,E2 -5674.817} C_VEL
LIN {X 0,Y 502.165,Z 348.319,A -85,B 0,C 180,E1 -5675.621,E2 -5675.621} C_VEL
LIN {X 0,Y 502.195,Z 345.99,A -85,B 0,C 180,E1 -5677.234,E2 -5677.234} C_VEL
LIN {X 0,Y 502.251,Z 343.11,A -85,B 0,C 180,E1 -5678.448,E2 -5678.448} C_VEL
LIN {X 0,Y 502.288,Z 339.193,A -85,B 0,C 180,E1 -5679.665,E2 -5679.665} C_VEL
LIN {X 0,Y 502.503,Z 333.124,A -85,B 0,C 180,E1 -5681.086,E2 -5681.086} C_VEL
LIN {X 0,Y 502.717,Z 326.464,A -85,B 0,C 180,E1 -5682.308,E2 -5682.308} C_VEL
LIN {X 0,Y 503.016,Z 318.165,A -85,B 0,C 180,E1 -5683.533,E2 -5683.533} C_VEL
LIN {X 0,Y 503.314,Z 309.581,A -85,B 0,C 180,E1 -5684.556,E2 -5684.556} C_VEL
LIN {X 0,Y 503.728,Z 299.404,A -85,B 0,C 180,E1 -5685.538,E2 -5685.538} C_VEL
LIN {X 0,Y 503.975,Z 289.777,A -85,B 0,C 180,E1 -5686.297,E2 -5686.297} C_VEL
LIN {X 0,Y 504.348,Z 278.407,A -85,B 0,C 180,E1 -5687.014,E2 -5687.014} C_VEL
LIN {X 0,Y 504.571,Z 266.724,A -85,B 0,C 180,E1 -5687.581,E2 -5687.581} C_VEL
LIN {X 0,Y 504.638,Z 257.224,A -85,B 0,C 180,E1 -5687.929,E2 -5687.929} C_VEL
LIN {X 0,Y 502.198,Z 246.424,A -85,B 0,C 180,E1 -5688.298,E2 -5688.298} C_VEL
LIN {X 0,Y 502.158,Z 242.933,A -85,B 0,C 180,E1 -5691.338,E2 -5691.338} C_VEL
LIN {X 0,Y 502.265,Z 239.304,A -85,B 0,C 180,E1 -5694.56,E2 -5694.56} C_VEL
LIN {X 0,Y 502.303,Z 236.125,A -85,B 0,C 180,E1 -5697.497,E2 -5697.497} C_VEL
LIN {X 0,Y 502.352,Z 233.192,A -85,B 0,C 180,E1 -5700.24,E2 -5700.24} C_VEL
LIN {X 0,Y 502.425,Z 230.229,A -85,B 0,C 180,E1 -5703.06,E2 -5703.06} C_VEL
LIN {X 0,Y 502.473,Z 227.185,A -85,B 0,C 180,E1 -5705.974,E2 -5705.974} C_VEL
LIN {X 0,Y 502.502,Z 225.994,A -85,B 0,C 180,E1 -5707.136,E2 -5707.136} C_VEL
LIN {X 0,Y 502.736,Z 225.86,A -85,B 0,C 180,E1 -5710.018,E2 -5710.018} C_VEL
LIN {X 0,Y 502.797,Z 225.854,A -85,B 0,C 180,E1 -5712.198,E2 -5712.198} C_VEL
LIN {X 0,Y 502.794,Z 225.854,A -85,B 0,C 180,E1 -5715.467,E2 -5715.467} C_VEL
LIN {X 0,Y 502.787,Z 225.858,A -85,B 0,C 180,E1 -5717.859,E2 -5717.859} C_VEL
LIN {X 0,Y 502.794,Z 225.858,A -85,B 0,C 180,E1 -5721.023,E2 -5721.023} C_VEL
LIN {X 0,Y 502.777,Z 225.859,A -85,B 0,C 180,E1 -5724.166,E2 -5724.166} C_VEL
LIN {X 0,Y 502.821,Z 225.85,A -85,B 0,C 180,E1 -5726.993,E2 -5726.993} C_VEL
LIN {X 0,Y 502.804,Z 225.851,A -85,B 0,C 180,E1 -5730.064,E2 -5730.064} C_VEL
LIN {X 0,Y 502.826,Z 225.852,A -85,B 0,C 180,E1 -5732.533,E2 -5732.533} C_VEL
LIN {X 0,Y 502.819,Z 225.851,A -85,B 0,C 180,E1 -5735.298,E2 -5735.298} C_VEL
LIN {X 0,Y 502.77,Z 225.858,A -85,B 0,C 180,E1 -5737.826,E2 -5737.826} C_VEL
LIN {X 0,Y 502.813,Z 225.853,A -85,B 0,C 180,E1 -5740.399,E2 -5740.399} C_VEL
LIN {X 0,Y 502.82,Z 225.85,A -85,B 0,C 180,E1 -5742.931,E2 -5742.931} C_VEL
LIN {X 0,Y 502.834,Z 225.851,A -85,B 0,C 180,E1 -5745.429,E2 -5745.429} C_VEL
LIN {X 0,Y 502.865,Z 225.847,A -85,B 0,C 180,E1 -5748.716,E2 -5748.716} C_VEL
LIN {X 0,Y 502.889,Z 225.844,A -85,B 0,C 180,E1 -5751.966,E2 -5751.966} C_VEL
LIN {X 0,Y 502.954,Z 225.834,A -85,B 0,C 180,E1 -5754.387,E2 -5754.387} C_VEL
LIN {X 0,Y 503.012,Z 225.827,A -85,B 0,C 180,E1 -5757.598,E2 -5757.598} C_VEL
LIN {X 0,Y 503.01,Z 225.827,A -85,B 0,C 180,E1 -5760,E2 -5760} C_VEL
LIN {X 0,Y 503.013,Z 225.828,A -85,B 0,C 180,E1 -5762.402,E2 -5762.402} C_VEL
LIN {X 0,Y 502.949,Z 225.837,A -85,B 0,C 180,E1 -5765.613,E2 -5765.613} C_VEL
LIN {X 0,Y 502.89,Z 225.841,A -85,B 0,C 180,E1 -5768.033,E2 -5768.033} C_VEL
LIN {X 0,Y 502.863,Z 225.844,A -85,B 0,C 180,E1 -5771.283,E2 -5771.283} C_VEL
LIN {X 0,Y 502.833,Z 225.847,A -85,B 0,C 180,E1 -5774.571,E2 -5774.571} C_VEL
LIN {X 0,Y 502.851,Z 225.846,A -85,B 0,C 180,E1 -5777.907,E2 -5777.907} C_VEL
LIN {X 0,Y 502.817,Z 225.853,A -85,B 0,C 180,E1 -5780.537,E2 -5780.537} C_VEL
LIN {X 0,Y 502.776,Z 225.856,A -85,B 0,C 180,E1 -5783.041,E2 -5783.041} C_VEL
LIN {X 0,Y 502.829,Z 225.85,A -85,B 0,C 180,E1 -5785.676,E2 -5785.676} C_VEL
LIN {X 0,Y 502.833,Z 225.853,A -85,B 0,C 180,E1 -5788.373,E2 -5788.373} C_VEL
LIN {X 0,Y 502.783,Z 225.857,A -85,B 0,C 180,E1 -5791.5,E2 -5791.5} C_VEL
LIN {X 0,Y 502.794,Z 225.854,A -85,B 0,C 180,E1 -5793.995,E2 -5793.995} C_VEL
LIN {X 0,Y 502.769,Z 225.857,A -85,B 0,C 180,E1 -5797.179,E2 -5797.179} C_VEL
LIN {X 0,Y 502.78,Z 225.86,A -85,B 0,C 180,E1 -5800.016,E2 -5800.016} C_VEL
LIN {X 0,Y 502.794,Z 225.854,A -85,B 0,C 180,E1 -5802.2,E2 -5802.2} C_VEL
LIN {X 0,Y 502.793,Z 225.856,A -85,B 0,C 180,E1 -5805.469,E2 -5805.469} C_VEL
LIN {X 0,Y 502.82,Z 225.854,A -85,B 0,C 180,E1 -5809.005,E2 -5809.005} C_VEL
LIN {X 0,Y 502.837,Z 225.969,A -85,B 0,C 180,E1 -5810.771,E2 -5810.771} C_VEL
LIN {X 0,Y 504.022,Z 232.921,A -85,B 0,C 180,E1 -5813.599,E2 -5813.599} C_VEL
LIN {X 0,Y 504.144,Z 237.6,A -85,B 0,C 180,E1 -5815.335,E2 -5815.335} C_VEL
LIN {X 0,Y 503.872,Z 245.957,A -85,B 0,C 180,E1 -5818.302,E2 -5818.302} C_VEL
LIN {X 0,Y 503.576,Z 254.49,A -85,B 0,C 180,E1 -5821.204,E2 -5821.204} C_VEL
LIN {X 0,Y 503.341,Z 262.686,A -85,B 0,C 180,E1 -5823.909,E2 -5823.909} C_VEL
LIN {X 0,Y 503.087,Z 272.229,A -85,B 0,C 180,E1 -5826.975,E2 -5826.975} C_VEL
LIN {X 0,Y 502.87,Z 281.496,A -85,B 0,C 180,E1 -5829.978,E2 -5829.978} C_VEL
LIN {X 0,Y 502.623,Z 290.764,A -85,B 0,C 180,E1 -5832.926,E2 -5832.926} C_VEL
LIN {X 0,Y 502.487,Z 299.576,A -85,B 0,C 180,E1 -5835.691,E2 -5835.691} C_VEL
LIN {X 0,Y 504.715,Z 313.141,A -85,B 0,C 180,E1 -5836.077,E2 -5836.077} C_VEL
LIN {X 0,Y 504.48,Z 325.011,A -85,B 0,C 180,E1 -5836.507,E2 -5836.507} C_VEL
LIN {X 0,Y 504.12,Z 335.431,A -85,B 0,C 180,E1 -5837.01,E2 -5837.01} C_VEL
LIN {X 0,Y 503.744,Z 347.419,A -85,B 0,C 180,E1 -5837.764,E2 -5837.764} C_VEL
LIN {X 0,Y 503.471,Z 358.278,A -85,B 0,C 180,E1 -5838.63,E2 -5838.63} C_VEL
LIN {X 0,Y 503.076,Z 367.551,A -85,B 0,C 180,E1 -5839.538,E2 -5839.538} C_VEL
LIN {X 0,Y 502.81,Z 376.001,A -85,B 0,C 180,E1 -5840.548,E2 -5840.548} C_VEL
LIN {X 0,Y 502.541,Z 384.244,A -85,B 0,C 180,E1 -5841.76,E2 -5841.76} C_VEL
LIN {X 0,Y 502.344,Z 390.883,A -85,B 0,C 180,E1 -5842.97,E2 -5842.97} C_VEL
LIN {X 0,Y 502.259,Z 396.954,A -85,B 0,C 180,E1 -5844.38,E2 -5844.38} C_VEL
LIN {X 0,Y 502.128,Z 400.898,A -85,B 0,C 180,E1 -5845.586,E2 -5845.586} C_VEL
LIN {X 0,Y 502.12,Z 403.81,A -85,B 0,C 180,E1 -5846.792,E2 -5846.792} C_VEL
LIN {X 0,Y 502.066,Z 405.197,A -85,B 0,C 180,E1 -5847.594,E2 -5847.594} C_VEL
LIN {X 0,Y 501.99,Z 406.786,A -85,B 0,C 180,E1 -5849.199,E2 -5849.199} C_VEL
LIN {X 0,Y 501.98,Z 407,A -85,B 0,C 180,E1 -5850.001,E2 -5850.001} C_VEL
LIN {X 0,Y 502.036,Z 406.184,A -85,B 0,C 180,E1 -5851.606,E2 -5851.606} C_VEL
LIN {X 0,Y 502.066,Z 405.196,A -85,B 0,C 180,E1 -5852.408,E2 -5852.408} C_VEL
LIN {X 0,Y 502.121,Z 403.808,A -85,B 0,C 180,E1 -5853.211,E2 -5853.211} C_VEL
LIN {X 0,Y 502.129,Z 400.892,A -85,B 0,C 180,E1 -5854.416,E2 -5854.416} C_VEL
LIN {X 0,Y 502.26,Z 396.944,A -85,B 0,C 180,E1 -5855.622,E2 -5855.622} C_VEL
LIN {X 0,Y 502.337,Z 390.971,A -85,B 0,C 180,E1 -5857.013,E2 -5857.013} C_VEL
LIN {X 0,Y 502.543,Z 384.229,A -85,B 0,C 180,E1 -5858.243,E2 -5858.243} C_VEL
LIN {X 0,Y 502.812,Z 375.983,A -85,B 0,C 180,E1 -5859.454,E2 -5859.454} C_VEL
LIN {X 0,Y 503.078,Z 367.529,A -85,B 0,C 180,E1 -5860.465,E2 -5860.465} C_VEL
LIN {X 0,Y 503.507,Z 357.081,A -85,B 0,C 180,E1 -5861.474,E2 -5861.474} C_VEL
LIN {X 0,Y 503.801,Z 345.369,A -85,B 0,C 180,E1 -5862.382,E2 -5862.382} C_VEL
LIN {X 0,Y 504.162,Z 333.468,A -85,B 0,C 180,E1 -5863.094,E2 -5863.094} C_VEL
LIN {X 0,Y 504.52,Z 321.138,A -85,B 0,C 180,E1 -5863.648,E2 -5863.648} C_VEL
LIN {X 0,Y 504.515,Z 312.135,A -85,B 0,C 180,E1 -5863.957,E2 -5863.957} C_VEL
LIN {X 0,Y 502.467,Z 299.527,A -85,B 0,C 180,E1 -5864.325,E2 -5864.325} C_VEL
LIN {X 0,Y 502.665,Z 289.432,A -85,B 0,C 180,E1 -5867.495,E2 -5867.495} C_VEL
LIN {X 0,Y 502.907,Z 279.826,A -85,B 0,C 180,E1 -5870.559,E2 -5870.559} C_VEL
LIN {X 0,Y 503.191,Z 269.574,A -85,B 0,C 180,E1 -5873.895,E2 -5873.895} C_VEL
LIN {X 0,Y 503.453,Z 259.899,A -85,B 0,C 180,E1 -5877.013,E2 -5877.013} C_VEL
LIN {X 0,Y 503.727,Z 250.476,A -85,B 0,C 180,E1 -5880.152,E2 -5880.152} C_VEL
LIN {X 0,Y 504.022,Z 241.646,A -85,B 0,C 180,E1 -5883.214,E2 -5883.214} C_VEL
LIN {X 0,Y 504.199,Z 234.422,A -85,B 0,C 180,E1 -5885.835,E2 -5885.835} C_VEL
LIN {X 0,Y 503.108,Z 227.574,A -85,B 0,C 180,E1 -5888.531,E2 -5888.531} C_VEL
LIN {X 0,Y 502.799,Z 225.858,A -85,B 0,C 180,E1 -5889.235,E2 -5889.235} C_VEL
LIN {X 0,Y 502.81,Z 225.857,A -85,B 0,C 180,E1 -5892.2,E2 -5892.2} C_VEL
LIN {X 0,Y 502.808,Z 225.856,A -85,B 0,C 180,E1 -5895.469,E2 -5895.469} C_VEL
LIN {X 0,Y 502.826,Z 225.852,A -85,B 0,C 180,E1 -5898.935,E2 -5898.935} C_VEL
LIN {X 0,Y 502.796,Z 225.852,A -85,B 0,C 180,E1 -5902.046,E2 -5902.046} C_VEL
LIN {X 0,Y 502.794,Z 225.854,A -85,B 0,C 180,E1 -5905.034,E2 -5905.034} C_VEL
LIN {X 0,Y 502.769,Z 225.857,A -85,B 0,C 180,E1 -5907.914,E2 -5907.914} C_VEL
LIN {X 0,Y 502.819,Z 225.85,A -85,B 0,C 180,E1 -5910.712,E2 -5910.712} C_VEL
LIN {X 0,Y 502.852,Z 225.849,A -85,B 0,C 180,E1 -5913.444,E2 -5913.444} C_VEL
LIN {X 0,Y 502.781,Z 225.855,A -85,B 0,C 180,E1 -5916.086,E2 -5916.086} C_VEL
LIN {X 0,Y 502.79,Z 225.858,A -85,B 0,C 180,E1 -5918.689,E2 -5918.689} C_VEL
LIN {X 0,Y 502.818,Z 225.851,A -85,B 0,C 180,E1 -5921.248,E2 -5921.248} C_VEL
LIN {X 0,Y 502.842,Z 225.847,A -85,B 0,C 180,E1 -5924.665,E2 -5924.665} C_VEL
LIN {X 0,Y 502.876,Z 225.845,A -85,B 0,C 180,E1 -5928.044,E2 -5928.044} C_VEL
LIN {X 0,Y 502.858,Z 225.848,A -85,B 0,C 180,E1 -5931.156,E2 -5931.156} C_VEL
LIN {X 0,Y 502.912,Z 225.84,A -85,B 0,C 180,E1 -5933.581,E2 -5933.581} C_VEL
LIN {X 0,Y 502.902,Z 225.843,A -85,B 0,C 180,E1 -5936.796,E2 -5936.796} C_VEL
LIN {X 0,Y 503.019,Z 225.826,A -85,B 0,C 180,E1 -5939.2,E2 -5939.2} C_VEL
LIN {X 0,Y 503.023,Z 225.826,A -85,B 0,C 180,E1 -5942.402,E2 -5942.402} C_VEL
LIN {X 0,Y 502.893,Z 225.844,A -85,B 0,C 180,E1 -5945.614,E2 -5945.614} C_VEL
LIN {X 0,Y 502.855,Z 225.844,A -85,B 0,C 180,E1 -5948.034,E2 -5948.034} C_VEL
LIN {X 0,Y 502.88,Z 225.844,A -85,B 0,C 180,E1 -5951.283,E2 -5951.283} C_VEL
LIN {X 0,Y 502.851,Z 225.851,A -85,B 0,C 180,E1 -5954.571,E2 -5954.571} C_VEL
LIN {X 0,Y 502.83,Z 225.852,A -85,B 0,C 180,E1 -5957.908,E2 -5957.908} C_VEL
LIN {X 0,Y 502.837,Z 225.848,A -85,B 0,C 180,E1 -5960.536,E2 -5960.536} C_VEL
LIN {X 0,Y 502.791,Z 225.858,A -85,B 0,C 180,E1 -5963.041,E2 -5963.041} C_VEL
LIN {X 0,Y 502.764,Z 225.856,A -85,B 0,C 180,E1 -5965.68,E2 -5965.68} C_VEL
LIN {X 0,Y 502.778,Z 225.858,A -85,B 0,C 180,E1 -5968.377,E2 -5968.377} C_VEL
LIN {X 0,Y 502.799,Z 225.852,A -85,B 0,C 180,E1 -5971.143,E2 -5971.143} C_VEL
LIN {X 0,Y 502.797,Z 225.857,A -85,B 0,C 180,E1 -5973.995,E2 -5973.995} C_VEL
LIN {X 0,Y 502.772,Z 225.859,A -85,B 0,C 180,E1 -5977.175,E2 -5977.175} C_VEL
LIN {X 0,Y 502.791,Z 225.854,A -85,B 0,C 180,E1 -5980.015,E2 -5980.015} C_VEL
LIN {X 0,Y 502.811,Z 225.852,A -85,B 0,C 180,E1 -5982.199,E2 -5982.199} C_VEL
LIN {X 0,Y 502.784,Z 225.853,A -85,B 0,C 180,E1 -5985.471,E2 -5985.471} C_VEL
LIN {X 0,Y 502.756,Z 225.856,A -85,B 0,C 180,E1 -5988.927,E2 -5988.927} C_VEL
LIN {X 0,Y 502.796,Z 225.855,A -85,B 0,C 180,E1 -5992.045,E2 -5992.045} C_VEL
LIN {X 0,Y 502.802,Z 225.855,A -85,B 0,C 180,E1 -5995.033,E2 -5995.033} C_VEL
LIN {X 0,Y 502.786,Z 225.856,A -85,B 0,C 180,E1 -5997.17,E2 -5997.17} C_VEL
LIN {X 0,Y 502.067,Z 225.945,A -85,B 0,C 180,E1 -5997.838,E2 -5997.838} C_VEL
LIN {X 0,Y 499.141,Z 226.311,A -85,B 0,C 180,E1 -5998.921,E2 -5998.921} C_VEL
LIN {X 0,Y 496.66,Z 226.623,A -85,B 0,C 180,E1 -5999.794,E2 -5999.794} C_VEL
LIN {X 0,Y 495.557,Z 226.759,A -85,B 0,C 180,E1 -6000.469,E2 -6000.469} C_VEL
LIN {X 0,Y 495.445,Z 226.772,A -85,B 0,C 180,E1 -6000.698,E2 -6000.698} C_VEL
LIN {X 0,Y 495.378,Z 226.991,A -85,B 0,C 180,E1 -6001.595,E2 -6001.595} C_VEL
LIN {X 0,Y 495.306,Z 230.402,A -85,B 0,C 180,E1 -6004.805,E2 -6004.805} C_VEL
LIN {X 0,Y 495.258,Z 233.258,A -85,B 0,C 180,E1 -6007.47,E2 -6007.47} C_VEL
LIN {X 0,Y 495.221,Z 236.066,A -85,B 0,C 180,E1 -6010.085,E2 -6010.085} C_VEL
LIN {X 0,Y 495.209,Z 238.874,A -85,B 0,C 180,E1 -6012.659,E2 -6012.659} C_VEL
LIN {X 0,Y 495.192,Z 241.709,A -85,B 0,C 180,E1 -6015.198,E2 -6015.198} C_VEL
LIN {X 0,Y 495.234,Z 245.536,A -85,B 0,C 180,E1 -6018.539,E2 -6018.539} C_VEL
LIN {X 0,Y 495.159,Z 246.783,A -85,B 0,C 180,E1 -6019.589,E2 -6019.589} C_VEL
LIN {X 0,Y 497.851,Z 259.322,A -85,B 0,C 180,E1 -6020.028,E2 -6020.028} C_VEL
LIN {X 0,Y 497.637,Z 272.166,A -85,B 0,C 180,E1 -6020.549,E2 -6020.549} C_VEL
LIN {X 0,Y 497.36,Z 283.292,A -85,B 0,C 180,E1 -6021.159,E2 -6021.159} C_VEL
LIN {X 0,Y 496.871,Z 294.892,A -85,B 0,C 180,E1 -6021.977,E2 -6021.977} C_VEL
LIN {X 0,Y 496.611,Z 305.121,A -85,B 0,C 180,E1 -6022.886,E2 -6022.886} C_VEL
LIN {X 0,Y 496.238,Z 314.451,A -85,B 0,C 180,E1 -6023.901,E2 -6023.901} C_VEL
LIN {X 0,Y 495.836,Z 323.439,A -85,B 0,C 180,E1 -6025.12,E2 -6025.12} C_VEL
LIN {X 0,Y 495.576,Z 330.679,A -85,B 0,C 180,E1 -6026.34,E2 -6026.34} C_VEL
LIN {X 0,Y 495.204,Z 336.51,A -85,B 0,C 180,E1 -6027.559,E2 -6027.559} C_VEL
LIN {X 0,Y 495.201,Z 341.092,A -85,B 0,C 180,E1 -6028.779,E2 -6028.779} C_VEL
LIN {X 0,Y 495.006,Z 344.615,A -85,B 0,C 180,E1 -6029.999,E2 -6029.999} C_VEL
LIN {X 0,Y 494.96,Z 346.424,A -85,B 0,C 180,E1 -6030.812,E2 -6030.812} C_VEL
LIN {X 0,Y 495.063,Z 348.736,A -85,B 0,C 180,E1 -6032.44,E2 -6032.44} C_VEL
LIN {X 0,Y 495.103,Z 349.321,A -85,B 0,C 180,E1 -6033.254,E2 -6033.254} C_VEL
LIN {X 0,Y 495.107,Z 349.521,A -85,B 0,C 180,E1 -6034.069,E2 -6034.069} C_VEL
LIN {X 0,Y 494.994,Z 349.302,A -85,B 0,C 180,E1 -6034.886,E2 -6034.886} C_VEL
LIN {X 0,Y 495.067,Z 347.838,A -85,B 0,C 180,E1 -6036.419,E2 -6036.419} C_VEL
LIN {X 0,Y 495.122,Z 346.303,A -85,B 0,C 180,E1 -6037.338,E2 -6037.338} C_VEL
LIN {X 0,Y 495.191,Z 343.381,A -85,B 0,C 180,E1 -6038.569,E2 -6038.569} C_VEL
LIN {X 0,Y 495.243,Z 339.413,A -85,B 0,C 180,E1 -6039.804,E2 -6039.804} C_VEL
LIN {X 0,Y 495.467,Z 333.267,A -85,B 0,C 180,E1 -6041.246,E2 -6041.246} C_VEL
LIN {X 0,Y 495.732,Z 326.542,A -85,B 0,C 180,E1 -6042.485,E2 -6042.485} C_VEL
LIN {X 0,Y 496.042,Z 318.149,A -85,B 0,C 180,E1 -6043.727,E2 -6043.727} C_VEL
LIN {X 0,Y 496.365,Z 309.452,A -85,B 0,C 180,E1 -6044.764,E2 -6044.764} C_VEL
LIN {X 0,Y 496.798,Z 299.971,A -85,B 0,C 180,E1 -6045.688,E2 -6045.688} C_VEL
LIN {X 0,Y 497.12,Z 289.398,A -85,B 0,C 180,E1 -6046.529,E2 -6046.529} C_VEL
LIN {X 0,Y 497.476,Z 277.804,A -85,B 0,C 180,E1 -6047.257,E2 -6047.257} C_VEL
LIN {X 0,Y 497.751,Z 265.24,A -85,B 0,C 180,E1 -6047.848,E2 -6047.848} C_VEL
LIN {X 0,Y 497.824,Z 258.569,A -85,B 0,C 180,E1 -6048.093,E2 -6048.093} C_VEL
LIN {X 0,Y 495.145,Z 246.828,A -85,B 0,C 180,E1 -6048.503,E2 -6048.503} C_VEL
LIN {X 0,Y 495.112,Z 243.224,A -85,B 0,C 180,E1 -6051.656,E2 -6051.656} C_VEL
LIN {X 0,Y 495.216,Z 239.788,A -85,B 0,C 180,E1 -6054.731,E2 -6054.731} C_VEL
LIN {X 0,Y 495.244,Z 237.338,A -85,B 0,C 180,E1 -6057.006,E2 -6057.006} C_VEL
LIN {X 0,Y 495.299,Z 234.097,A -85,B 0,C 180,E1 -6060.053,E2 -6060.053} C_VEL
LIN {X 0,Y 495.359,Z 230.853,A -85,B 0,C 180,E1 -6063.167,E2 -6063.167} C_VEL
LIN {X 0,Y 495.42,Z 227.895,A -85,B 0,C 180,E1 -6066.04,E2 -6066.04} C_VEL
LIN {X 0,Y 495.477,Z 226.77,A -85,B 0,C 180,E1 -6067.582,E2 -6067.582} C_VEL
LIN {X 0,Y 495.71,Z 226.735,A -85,B 0,C 180,E1 -6070.04,E2 -6070.04} C_VEL
LIN {X 0,Y 495.72,Z 226.738,A -85,B 0,C 180,E1 -6072.882,E2 -6072.882} C_VEL
LIN {X 0,Y 495.723,Z 226.739,A -85,B 0,C 180,E1 -6075.997,E2 -6075.997} C_VEL
LIN {X 0,Y 495.745,Z 226.736,A -85,B 0,C 180,E1 -6079.298,E2 -6079.298} C_VEL
LIN {X 0,Y 495.724,Z 226.738,A -85,B 0,C 180,E1 -6082.438,E2 -6082.438} C_VEL
LIN {X 0,Y 495.769,Z 226.73,A -85,B 0,C 180,E1 -6085.456,E2 -6085.456} C_VEL
LIN {X 0,Y 495.744,Z 226.731,A -85,B 0,C 180,E1 -6088.363,E2 -6088.363} C_VEL
LIN {X 0,Y 495.778,Z 226.727,A -85,B 0,C 180,E1 -6091.506,E2 -6091.506} C_VEL
LIN {X 0,Y 495.79,Z 226.728,A -85,B 0,C 180,E1 -6093.932,E2 -6093.932} C_VEL
LIN {X 0,Y 495.751,Z 226.733,A -85,B 0,C 180,E1 -6097.138,E2 -6097.138} C_VEL
LIN {X 0,Y 495.759,Z 226.729,A -85,B 0,C 180,E1 -6100.109,E2 -6100.109} C_VEL
LIN {X 0,Y 495.771,Z 226.73,A -85,B 0,C 180,E1 -6102.681,E2 -6102.681} C_VEL
LIN {X 0,Y 495.779,Z 226.728,A -85,B 0,C 180,E1 -6105.217,E2 -6105.217} C_VEL
LIN {X 0,Y 495.84,Z 226.721,A -85,B 0,C 180,E1 -6108.554,E2 -6108.554} C_VEL
LIN {X 0,Y 495.86,Z 226.718,A -85,B 0,C 180,E1 -6111.852,E2 -6111.852} C_VEL
LIN {X 0,Y 495.908,Z 226.712,A -85,B 0,C 180,E1 -6114.307,E2 -6114.307} C_VEL
LIN {X 0,Y 495.981,Z 226.703,A -85,B 0,C 180,E1 -6117.564,E2 -6117.564} C_VEL
LIN {X 0,Y 495.969,Z 226.706,A -85,B 0,C 180,E1 -6120.812,E2 -6120.812} C_VEL
LIN {X 0,Y 495.982,Z 226.704,A -85,B 0,C 180,E1 -6122.436,E2 -6122.436} C_VEL
LIN {X 0,Y 495.903,Z 226.714,A -85,B 0,C 180,E1 -6125.693,E2 -6125.693} C_VEL
LIN {X 0,Y 495.861,Z 226.717,A -85,B 0,C 180,E1 -6128.148,E2 -6128.148} C_VEL
LIN {X 0,Y 495.838,Z 226.719,A -85,B 0,C 180,E1 -6131.445,E2 -6131.445} C_VEL
LIN {X 0,Y 495.778,Z 226.727,A -85,B 0,C 180,E1 -6134.783,E2 -6134.783} C_VEL
LIN {X 0,Y 495.778,Z 226.729,A -85,B 0,C 180,E1 -6137.319,E2 -6137.319} C_VEL
LIN {X 0,Y 495.761,Z 226.73,A -85,B 0,C 180,E1 -6139.891,E2 -6139.891} C_VEL
LIN {X 0,Y 495.747,Z 226.731,A -85,B 0,C 180,E1 -6142.861,E2 -6142.861} C_VEL
LIN {X 0,Y 495.788,Z 226.726,A -85,B 0,C 180,E1 -6146.068,E2 -6146.068} C_VEL
LIN {X 0,Y 495.771,Z 226.73,A -85,B 0,C 180,E1 -6148.815,E2 -6148.815} C_VEL
LIN {X 0,Y 495.746,Z 226.736,A -85,B 0,C 180,E1 -6151.726,E2 -6151.726} C_VEL
LIN {X 0,Y 495.759,Z 226.732,A -85,B 0,C 180,E1 -6154.695,E2 -6154.695} C_VEL
LIN {X 0,Y 495.72,Z 226.733,A -85,B 0,C 180,E1 -6157.563,E2 -6157.563} C_VEL
LIN {X 0,Y 495.757,Z 226.73,A -85,B 0,C 180,E1 -6160.701,E2 -6160.701} C_VEL
LIN {X 0,Y 495.722,Z 226.735,A -85,B 0,C 180,E1 -6164.002,E2 -6164.002} C_VEL
LIN {X 0,Y 495.719,Z 226.738,A -85,B 0,C 180,E1 -6167.118,E2 -6167.118} C_VEL
LIN {X 0,Y 495.783,Z 226.733,A -85,B 0,C 180,E1 -6169.95,E2 -6169.95} C_VEL
LIN {X 0,Y 495.791,Z 226.845,A -85,B 0,C 180,E1 -6170.479,E2 -6170.479} C_VEL
LIN {X 0,Y 496.863,Z 232.98,A -85,B 0,C 180,E1 -6173.049,E2 -6173.049} C_VEL
LIN {X 0,Y 497.21,Z 236.914,A -85,B 0,C 180,E1 -6174.584,E2 -6174.584} C_VEL
LIN {X 0,Y 496.961,Z 244.949,A -85,B 0,C 180,E1 -6177.495,E2 -6177.495} C_VEL
LIN {X 0,Y 496.609,Z 252.947,A -85,B 0,C 180,E1 -6180.311,E2 -6180.311} C_VEL
LIN {X 0,Y 496.406,Z 261.279,A -85,B 0,C 180,E1 -6183.118,E2 -6183.118} C_VEL
LIN {X 0,Y 496.115,Z 270.672,A -85,B 0,C 180,E1 -6186.19,E2 -6186.19} C_VEL
LIN {X 0,Y 495.89,Z 280.297,A -85,B 0,C 180,E1 -6189.291,E2 -6189.291} C_VEL
LIN {X 0,Y 495.635,Z 289.44,A -85,B 0,C 180,E1 -6192.251,E2 -6192.251} C_VEL
LIN {X 0,Y 495.412,Z 299.616,A -85,B 0,C 180,E1 -6195.486,E2 -6195.486} C_VEL
LIN {X 0,Y 497.69,Z 313.141,A -85,B 0,C 180,E1 -6195.877,E2 -6195.877} C_VEL
LIN {X 0,Y 497.554,Z 326.14,A -85,B 0,C 180,E1 -6196.368,E2 -6196.368} C_VEL
LIN {X 0,Y 497.166,Z 337.195,A -85,B 0,C 180,E1 -6196.929,E2 -6196.929} C_VEL
LIN {X 0,Y 496.759,Z 348.317,A -85,B 0,C 180,E1 -6197.655,E2 -6197.655} C_VEL
LIN {X 0,Y 496.438,Z 359.413,A -85,B 0,C 180,E1 -6198.57,E2 -6198.57} C_VEL
LIN {X 0,Y 496.005,Z 369.345,A -85,B 0,C 180,E1 -6199.593,E2 -6199.593} C_VEL
LIN {X 0,Y 495.672,Z 378.969,A -85,B 0,C 180,E1 -6200.823,E2 -6200.823} C_VEL
LIN {X 0,Y 495.402,Z 386.629,A -85,B 0,C 180,E1 -6202.051,E2 -6202.051} C_VEL
LIN {X 0,Y 495.202,Z 393.685,A -85,B 0,C 180,E1 -6203.482,E2 -6203.482} C_VEL
LIN {X 0,Y 495.122,Z 398.377,A -85,B 0,C 180,E1 -6204.707,E2 -6204.707} C_VEL
LIN {X 0,Y 495.049,Z 401.961,A -85,B 0,C 180,E1 -6205.931,E2 -6205.931} C_VEL
LIN {X 0,Y 495.042,Z 403.81,A -85,B 0,C 180,E1 -6206.746,E2 -6206.746} C_VEL
LIN {X 0,Y 494.961,Z 406.184,A -85,B 0,C 180,E1 -6208.374,E2 -6208.374} C_VEL
LIN {X 0,Y 494.898,Z 407,A -85,B 0,C 180,E1 -6210.001,E2 -6210.001} C_VEL
LIN {X 0,Y 494.961,Z 406.183,A -85,B 0,C 180,E1 -6211.628,E2 -6211.628} C_VEL
LIN {X 0,Y 495.043,Z 403.808,A -85,B 0,C 180,E1 -6213.257,E2 -6213.257} C_VEL
LIN {X 0,Y 495.029,Z 400.892,A -85,B 0,C 180,E1 -6214.48,E2 -6214.48} C_VEL
LIN {X 0,Y 495.211,Z 395.798,A -85,B 0,C 180,E1 -6216,E2 -6216} C_VEL
LIN {X 0,Y 495.279,Z 389.863,A -85,B 0,C 180,E1 -6217.338,E2 -6217.338} C_VEL
LIN {X 0,Y 495.557,Z 382.996,A -85,B 0,C 180,E1 -6218.565,E2 -6218.565} C_VEL
LIN {X 0,Y 495.848,Z 374.404,A -85,B 0,C 180,E1 -6219.794,E2 -6219.794} C_VEL
LIN {X 0,Y 496.199,Z 365.588,A -85,B 0,C 180,E1 -6220.818,E2 -6220.818} C_VEL
LIN {X 0,Y 496.582,Z 354.731,A -85,B 0,C 180,E1 -6221.843,E2 -6221.843} C_VEL
LIN {X 0,Y 496.903,Z 344.161,A -85,B 0,C 180,E1 -6222.639,E2 -6222.639} C_VEL
LIN {X 0,Y 497.293,Z 331.478,A -85,B 0,C 180,E1 -6223.382,E2 -6223.382} C_VEL
LIN {X 0,Y 497.649,Z 319.837,A -85,B 0,C 180,E1 -6223.892,E2 -6223.892} C_VEL
LIN {X 0,Y 497.575,Z 312.591,A -85,B 0,C 180,E1 -6224.142,E2 -6224.142} C_VEL
LIN {X 0,Y 495.425,Z 299.527,A -85,B 0,C 180,E1 -6224.533,E2 -6224.533} C_VEL
LIN {X 0,Y 495.64,Z 289.432,A -85,B 0,C 180,E1 -6227.751,E2 -6227.751} C_VEL
LIN {X 0,Y 495.889,Z 280.165,A -85,B 0,C 180,E1 -6230.752,E2 -6230.752} C_VEL
LIN {X 0,Y 496.122,Z 270.671,A -85,B 0,C 180,E1 -6233.813,E2 -6233.813} C_VEL
LIN {X 0,Y 496.42,Z 261.117,A -85,B 0,C 180,E1 -6236.94,E2 -6236.94} C_VEL
LIN {X 0,Y 496.619,Z 252.995,A -85,B 0,C 180,E1 -6239.691,E2 -6239.691} C_VEL
LIN {X 0,Y 496.965,Z 244.908,A -85,B 0,C 180,E1 -6242.507,E2 -6242.507} C_VEL
LIN {X 0,Y 497.221,Z 236.931,A -85,B 0,C 180,E1 -6245.418,E2 -6245.418} C_VEL
LIN {X 0,Y 496.854,Z 232.937,A -85,B 0,C 180,E1 -6246.954,E2 -6246.954} C_VEL
LIN {X 0,Y 495.747,Z 226.735,A -85,B 0,C 180,E1 -6249.528,E2 -6249.528} C_VEL
LIN {X 0,Y 495.744,Z 226.737,A -85,B 0,C 180,E1 -6252.508,E2 -6252.508} C_VEL
LIN {X 0,Y 495.756,Z 226.733,A -85,B 0,C 180,E1 -6255.14,E2 -6255.14} C_VEL
LIN {X 0,Y 495.763,Z 226.73,A -85,B 0,C 180,E1 -6258.219,E2 -6258.219} C_VEL
LIN {X 0,Y 495.753,Z 226.732,A -85,B 0,C 180,E1 -6261.409,E2 -6261.409} C_VEL
LIN {X 0,Y 495.745,Z 226.734,A -85,B 0,C 180,E1 -6264.462,E2 -6264.462} C_VEL
LIN {X 0,Y 495.748,Z 226.73,A -85,B 0,C 180,E1 -6267.404,E2 -6267.404} C_VEL
LIN {X 0,Y 495.768,Z 226.732,A -85,B 0,C 180,E1 -6270.254,E2 -6270.254} C_VEL
LIN {X 0,Y 495.782,Z 226.729,A -85,B 0,C 180,E1 -6273.262,E2 -6273.262} C_VEL
LIN {X 0,Y 495.73,Z 226.736,A -85,B 0,C 180,E1 -6275.724,E2 -6275.724} C_VEL
LIN {X 0,Y 495.749,Z 226.733,A -85,B 0,C 180,E1 -6278.371,E2 -6278.371} C_VEL
LIN {X 0,Y 495.778,Z 226.729,A -85,B 0,C 180,E1 -6280.971,E2 -6280.971} C_VEL
LIN {X 0,Y 495.809,Z 226.724,A -85,B 0,C 180,E1 -6284.558,E2 -6284.558} C_VEL
LIN {X 0,Y 495.828,Z 226.724,A -85,B 0,C 180,E1 -6287.97,E2 -6287.97} C_VEL
LIN {X 0,Y 495.812,Z 226.725,A -85,B 0,C 180,E1 -6291.03,E2 -6291.03} C_VEL
LIN {X 0,Y 495.867,Z 226.719,A -85,B 0,C 180,E1 -6293.49,E2 -6293.49} C_VEL
LIN {X 0,Y 495.846,Z 226.722,A -85,B 0,C 180,E1 -6296.75,E2 -6296.75} C_VEL
LIN {X 0,Y 495.875,Z 226.718,A -85,B 0,C 180,E1 -6298.376,E2 -6298.376} C_VEL
LIN {X 0,Y 495.95,Z 226.706,A -85,B 0,C 180,E1 -6300.812,E2 -6300.812} C_VEL
LIN {X 0,Y 495.991,Z 226.701,A -85,B 0,C 180,E1 -6302.436,E2 -6302.436} C_VEL
LIN {X 0,Y 495.85,Z 226.72,A -85,B 0,C 180,E1 -6305.694,E2 -6305.694} C_VEL
LIN {X 0,Y 495.82,Z 226.721,A -85,B 0,C 180,E1 -6308.149,E2 -6308.149} C_VEL
LIN {X 0,Y 495.856,Z 226.718,A -85,B 0,C 180,E1 -6311.445,E2 -6311.445} C_VEL
LIN {X 0,Y 495.797,Z 226.727,A -85,B 0,C 180,E1 -6314.783,E2 -6314.783} C_VEL
LIN {X 0,Y 495.771,Z 226.73,A -85,B 0,C 180,E1 -6317.319,E2 -6317.319} C_VEL
LIN {X 0,Y 495.777,Z 226.73,A -85,B 0,C 180,E1 -6319.89,E2 -6319.89} C_VEL
LIN {X 0,Y 495.765,Z 226.731,A -85,B 0,C 180,E1 -6322.86,E2 -6322.86} C_VEL
LIN {X 0,Y 495.711,Z 226.734,A -85,B 0,C 180,E1 -6326.073,E2 -6326.073} C_VEL
LIN {X 0,Y 495.733,Z 226.735,A -85,B 0,C 180,E1 -6328.818,E2 -6328.818} C_VEL
LIN {X 0,Y 495.761,Z 226.731,A -85,B 0,C 180,E1 -6331.725,E2 -6331.725} C_VEL
LIN {X 0,Y 495.769,Z 226.729,A -85,B 0,C 180,E1 -6334.692,E2 -6334.692} C_VEL
LIN {X 0,Y 495.729,Z 226.736,A -85,B 0,C 180,E1 -6337.562,E2 -6337.562} C_VEL
LIN {X 0,Y 495.763,Z 226.73,A -85,B 0,C 180,E1 -6340.046,E2 -6340.046} C_VEL
LIN {X 0,Y 495.722,Z 226.736,A -85,B 0,C 180,E1 -6342.884,E2 -6342.884} C_VEL
LIN {X 0,Y 495.719,Z 226.737,A -85,B 0,C 180,E1 -6345.996,E2 -6345.996} C_VEL
LIN {X 0,Y 495.716,Z 226.734,A -85,B 0,C 180,E1 -6349.294,E2 -6349.294} C_VEL
LIN {X 0,Y 495.75,Z 226.733,A -85,B 0,C 180,E1 -6351.407,E2 -6351.407} C_VEL
LIN {X 0,Y 495.752,Z 226.731,A -85,B 0,C 180,E1 -6354.461,E2 -6354.461} C_VEL
LIN {X 0,Y 495.743,Z 226.734,A -85,B 0,C 180,E1 -6357.403,E2 -6357.403} C_VEL
LIN {X 0,Y 495.526,Z 226.763,A -85,B 0,C 180,E1 -6360.237,E2 -6360.237} C_VEL
LIN {X 0,Y 495.445,Z 226.772,A -85,B 0,C 180,E1 -6360.698,E2 -6360.698} C_VEL
LIN {X 0,Y 494.705,Z 227.054,A -85,B 0,C 180,E1 -6361.375,E2 -6361.375} C_VEL
LIN {X 0,Y 491.78,Z 228.274,A -85,B 0,C 180,E1 -6362.467,E2 -6362.467} C_VEL
LIN {X 0,Y 489.345,Z 229.449,A -85,B 0,C 180,E1 -6363.345,E2 -6363.345} C_VEL
LIN {X 0,Y 488.308,Z 230.269,A -85,B 0,C 180,E1 -6364.024,E2 -6364.024} C_VEL
LIN {X 0,Y 488.226,Z 230.52,A -85,B 0,C 180,E1 -6364.255,E2 -6364.255} C_VEL
LIN {X 0,Y 488.205,Z 233.579,A -85,B 0,C 180,E1 -6367.126,E2 -6367.126} C_VEL
LIN {X 0,Y 488.186,Z 236.409,A -85,B 0,C 180,E1 -6369.786,E2 -6369.786} C_VEL
LIN {X 0,Y 488.157,Z 239.236,A -85,B 0,C 180,E1 -6372.401,E2 -6372.401} C_VEL
LIN {X 0,Y 488.141,Z 242.107,A -85,B 0,C 180,E1 -6374.979,E2 -6374.979} C_VEL
LIN {X 0,Y 488.164,Z 245.983,A -85,B 0,C 180,E1 -6378.371,E2 -6378.371} C_VEL
LIN {X 0,Y 488.119,Z 247.304,A -85,B 0,C 180,E1 -6379.394,E2 -6379.394} C_VEL
LIN {X 0,Y 490.948,Z 260.173,A -85,B 0,C 180,E1 -6379.847,E2 -6379.847} C_VEL
LIN {X 0,Y 490.761,Z 272.632,A -85,B 0,C 180,E1 -6380.364,E2 -6380.364} C_VEL
LIN {X 0,Y 490.423,Z 284.539,A -85,B 0,C 180,E1 -6381.033,E2 -6381.033} C_VEL
LIN {X 0,Y 489.913,Z 295.988,A -85,B 0,C 180,E1 -6381.862,E2 -6381.862} C_VEL
LIN {X 0,Y 489.627,Z 306.115,A -85,B 0,C 180,E1 -6382.784,E2 -6382.784} C_VEL
LIN {X 0,Y 489.247,Z 315.325,A -85,B 0,C 180,E1 -6383.814,E2 -6383.814} C_VEL
LIN {X 0,Y 488.82,Z 324.232,A -85,B 0,C 180,E1 -6385.05,E2 -6385.05} C_VEL
LIN {X 0,Y 488.517,Z 331.414,A -85,B 0,C 180,E1 -6386.287,E2 -6386.287} C_VEL
LIN {X 0,Y 488.144,Z 337.186,A -85,B 0,C 180,E1 -6387.523,E2 -6387.523} C_VEL
LIN {X 0,Y 488.131,Z 341.716,A -85,B 0,C 180,E1 -6388.761,E2 -6388.761} C_VEL
LIN {X 0,Y 487.926,Z 345.19,A -85,B 0,C 180,E1 -6389.999,E2 -6389.999} C_VEL
LIN {X 0,Y 487.88,Z 346.954,A -85,B 0,C 180,E1 -6390.824,E2 -6390.824} C_VEL
LIN {X 0,Y 488,Z 349.217,A -85,B 0,C 180,E1 -6392.475,E2 -6392.475} C_VEL
LIN {X 0,Y 488.024,Z 349.781,A -85,B 0,C 180,E1 -6393.301,E2 -6393.301} C_VEL
LIN {X 0,Y 488.021,Z 349.939,A -85,B 0,C 180,E1 -6394.128,E2 -6394.128} C_VEL
LIN {X 0,Y 488.015,Z 349.061,A -85,B 0,C 180,E1 -6395.784,E2 -6395.784} C_VEL
LIN {X 0,Y 488.022,Z 348.049,A -85,B 0,C 180,E1 -6396.614,E2 -6396.614} C_VEL
LIN {X 0,Y 488.052,Z 346.607,A -85,B 0,C 180,E1 -6397.445,E2 -6397.445} C_VEL
LIN {X 0,Y 488.117,Z 343.643,A -85,B 0,C 180,E1 -6398.694,E2 -6398.694} C_VEL
LIN {X 0,Y 488.196,Z 339.623,A -85,B 0,C 180,E1 -6399.946,E2 -6399.946} C_VEL
LIN {X 0,Y 488.448,Z 333.414,A -85,B 0,C 180,E1 -6401.409,E2 -6401.409} C_VEL
LIN {X 0,Y 488.736,Z 326.631,A -85,B 0,C 180,E1 -6402.666,E2 -6402.666} C_VEL
LIN {X 0,Y 489.089,Z 318.134,A -85,B 0,C 180,E1 -6403.926,E2 -6403.926} C_VEL
LIN {X 0,Y 489.423,Z 309.355,A -85,B 0,C 180,E1 -6404.978,E2 -6404.978} C_VEL
LIN {X 0,Y 489.87,Z 298.781,A -85,B 0,C 180,E1 -6406.006,E2 -6406.006} C_VEL
LIN {X 0,Y 490.246,Z 289.077,A -85,B 0,C 180,E1 -6406.767,E2 -6406.767} C_VEL
LIN {X 0,Y 490.604,Z 277.202,A -85,B 0,C 180,E1 -6407.506,E2 -6407.506} C_VEL
LIN {X 0,Y 490.926,Z 264.403,A -85,B 0,C 180,E1 -6408.102,E2 -6408.102} C_VEL
LIN {X 0,Y 490.858,Z 259.225,A -85,B 0,C 180,E1 -6408.295,E2 -6408.295} C_VEL
LIN {X 0,Y 488.047,Z 247.233,A -85,B 0,C 180,E1 -6408.725,E2 -6408.725} C_VEL
LIN {X 0,Y 488.017,Z 244.516,A -85,B 0,C 180,E1 -6411.1,E2 -6411.1} C_VEL
LIN {X 0,Y 488.089,Z 241.545,A -85,B 0,C 180,E1 -6413.775,E2 -6413.775} C_VEL
LIN {X 0,Y 488.205,Z 238.569,A -85,B 0,C 180,E1 -6416.503,E2 -6416.503} C_VEL
LIN {X 0,Y 488.213,Z 235.604,A -85,B 0,C 180,E1 -6419.302,E2 -6419.302} C_VEL
LIN {X 0,Y 488.247,Z 232.625,A -85,B 0,C 180,E1 -6422.179,E2 -6422.179} C_VEL
LIN {X 0,Y 488.35,Z 229.574,A -85,B 0,C 180,E1 -6425.144,E2 -6425.144} C_VEL
LIN {X 0,Y 488.379,Z 227.655,A -85,B 0,C 180,E1 -6427.184,E2 -6427.184} C_VEL
LIN {X 0,Y 488.624,Z 227.622,A -85,B 0,C 180,E1 -6429.26,E2 -6429.26} C_VEL
LIN {X 0,Y 488.693,Z 227.61,A -85,B 0,C 180,E1 -6431.597,E2 -6431.597} C_VEL
LIN {X 0,Y 488.706,Z 227.61,A -85,B 0,C 180,E1 -6434.8,E2 -6434.8} C_VEL
LIN {X 0,Y 488.68,Z 227.615,A -85,B 0,C 180,E1 -6437.473,E2 -6437.473} C_VEL
LIN {X 0,Y 488.693,Z 227.613,A -85,B 0,C 180,E1 -6440.745,E2 -6440.745} C_VEL
LIN {X 0,Y 488.677,Z 227.612,A -85,B 0,C 180,E1 -6443.868,E2 -6443.868} C_VEL
LIN {X 0,Y 488.726,Z 227.605,A -85,B 0,C 180,E1 -6446.876,E2 -6446.876} C_VEL
LIN {X 0,Y 488.713,Z 227.607,A -85,B 0,C 180,E1 -6449.78,E2 -6449.78} C_VEL
LIN {X 0,Y 488.789,Z 227.597,A -85,B 0,C 180,E1 -6453.054,E2 -6453.054} C_VEL
LIN {X 0,Y 488.683,Z 227.612,A -85,B 0,C 180,E1 -6456.254,E2 -6456.254} C_VEL
LIN {X 0,Y 488.735,Z 227.608,A -85,B 0,C 180,E1 -6459.175,E2 -6459.175} C_VEL
LIN {X 0,Y 488.719,Z 227.612,A -85,B 0,C 180,E1 -6462.423,E2 -6462.423} C_VEL
LIN {X 0,Y 488.751,Z 227.602,A -85,B 0,C 180,E1 -6464.999,E2 -6464.999} C_VEL
LIN {X 0,Y 488.794,Z 227.597,A -85,B 0,C 180,E1 -6468.387,E2 -6468.387} C_VEL
LIN {X 0,Y 488.803,Z 227.596,A -85,B 0,C 180,E1 -6471.733,E2 -6471.733} C_VEL
LIN {X 0,Y 488.864,Z 227.591,A -85,B 0,C 180,E1 -6474.224,E2 -6474.224} C_VEL
LIN {X 0,Y 488.949,Z 227.579,A -85,B 0,C 180,E1 -6477.528,E2 -6477.528} C_VEL
LIN {X 0,Y 488.92,Z 227.584,A -85,B 0,C 180,E1 -6480.824,E2 -6480.824} C_VEL
LIN {X 0,Y 488.95,Z 227.58,A -85,B 0,C 180,E1 -6482.471,E2 -6482.471} C_VEL
LIN {X 0,Y 488.86,Z 227.591,A -85,B 0,C 180,E1 -6485.776,E2 -6485.776} C_VEL
LIN {X 0,Y 488.805,Z 227.597,A -85,B 0,C 180,E1 -6488.267,E2 -6488.267} C_VEL
LIN {X 0,Y 488.793,Z 227.598,A -85,B 0,C 180,E1 -6491.613,E2 -6491.613} C_VEL
LIN {X 0,Y 488.75,Z 227.604,A -85,B 0,C 180,E1 -6495.001,E2 -6495.001} C_VEL
LIN {X 0,Y 488.744,Z 227.607,A -85,B 0,C 180,E1 -6498.443,E2 -6498.443} C_VEL
LIN {X 0,Y 488.695,Z 227.609,A -85,B 0,C 180,E1 -6501.071,E2 -6501.071} C_VEL
LIN {X 0,Y 488.672,Z 227.615,A -85,B 0,C 180,E1 -6503.747,E2 -6503.747} C_VEL
LIN {X 0,Y 488.789,Z 227.602,A -85,B 0,C 180,E1 -6506.946,E2 -6506.946} C_VEL
LIN {X 0,Y 488.709,Z 227.611,A -85,B 0,C 180,E1 -6510.365,E2 -6510.365} C_VEL
LIN {X 0,Y 488.724,Z 227.611,A -85,B 0,C 180,E1 -6513.485,E2 -6513.485} C_VEL
LIN {X 0,Y 488.673,Z 227.614,A -85,B 0,C 180,E1 -6516.355,E2 -6516.355} C_VEL
LIN {X 0,Y 488.693,Z 227.61,A -85,B 0,C 180,E1 -6519.255,E2 -6519.255} C_VEL
LIN {X 0,Y 488.698,Z 227.613,A -85,B 0,C 180,E1 -6521.601,E2 -6521.601} C_VEL
LIN {X 0,Y 488.704,Z 227.613,A -85,B 0,C 180,E1 -6524.803,E2 -6524.803} C_VEL
LIN {X 0,Y 488.685,Z 227.613,A -85,B 0,C 180,E1 -6527.476,E2 -6527.476} C_VEL
LIN {X 0,Y 488.749,Z 227.661,A -85,B 0,C 180,E1 -6530.151,E2 -6530.151} C_VEL
LIN {X 0,Y 489.881,Z 234.189,A -85,B 0,C 180,E1 -6532.949,E2 -6532.949} C_VEL
LIN {X 0,Y 490.242,Z 237.951,A -85,B 0,C 180,E1 -6534.448,E2 -6534.448} C_VEL
LIN {X 0,Y 490.005,Z 244.733,A -85,B 0,C 180,E1 -6536.975,E2 -6536.975} C_VEL
LIN {X 0,Y 489.677,Z 252.791,A -85,B 0,C 180,E1 -6539.847,E2 -6539.847} C_VEL
LIN {X 0,Y 489.408,Z 261.673,A -85,B 0,C 180,E1 -6542.915,E2 -6542.915} C_VEL
LIN {X 0,Y 489.053,Z 271.739,A -85,B 0,C 180,E1 -6546.275,E2 -6546.275} C_VEL
LIN {X 0,Y 488.825,Z 281.74,A -85,B 0,C 180,E1 -6549.481,E2 -6549.481} C_VEL
LIN {X 0,Y 488.561,Z 290.764,A -85,B 0,C 180,E1 -6552.418,E2 -6552.418} C_VEL
LIN {X 0,Y 488.371,Z 299.618,A -85,B 0,C 180,E1 -6555.272,E2 -6555.272} C_VEL
LIN {X 0,Y 490.563,Z 312.686,A -85,B 0,C 180,E1 -6555.654,E2 -6555.654} C_VEL
LIN {X 0,Y 490.863,Z 316.255,A -85,B 0,C 180,E1 -6555.782,E2 -6555.782} C_VEL
LIN {X 0,Y 490.471,Z 329.515,A -85,B 0,C 180,E1 -6556.325,E2 -6556.325} C_VEL
LIN {X 0,Y 490.117,Z 340.531,A -85,B 0,C 180,E1 -6556.941,E2 -6556.941} C_VEL
LIN {X 0,Y 489.752,Z 350.919,A -85,B 0,C 180,E1 -6557.676,E2 -6557.676} C_VEL
LIN {X 0,Y 489.371,Z 361.55,A -85,B 0,C 180,E1 -6558.612,E2 -6558.612} C_VEL
LIN {X 0,Y 488.953,Z 371.124,A -85,B 0,C 180,E1 -6559.651,E2 -6559.651} C_VEL
LIN {X 0,Y 488.656,Z 378.969,A -85,B 0,C 180,E1 -6560.69,E2 -6560.69} C_VEL
LIN {X 0,Y 488.36,Z 386.628,A -85,B 0,C 180,E1 -6561.935,E2 -6561.935} C_VEL
LIN {X 0,Y 488.14,Z 393.685,A -85,B 0,C 180,E1 -6563.387,E2 -6563.387} C_VEL
LIN {X 0,Y 488.06,Z 398.377,A -85,B 0,C 180,E1 -6564.631,E2 -6564.631} C_VEL
LIN {X 0,Y 487.947,Z 401.961,A -85,B 0,C 180,E1 -6565.871,E2 -6565.871} C_VEL
LIN {X 0,Y 487.966,Z 403.809,A -85,B 0,C 180,E1 -6566.699,E2 -6566.699} C_VEL
LIN {X 0,Y 487.889,Z 406.184,A -85,B 0,C 180,E1 -6568.35,E2 -6568.35} C_VEL
LIN {X 0,Y 487.819,Z 407,A -85,B 0,C 180,E1 -6570.001,E2 -6570.001} C_VEL
LIN {X 0,Y 487.889,Z 406.183,A -85,B 0,C 180,E1 -6571.652,E2 -6571.652} C_VEL
LIN {X 0,Y 487.967,Z 403.808,A -85,B 0,C 180,E1 -6573.304,E2 -6573.304} C_VEL
LIN {X 0,Y 487.938,Z 400.892,A -85,B 0,C 180,E1 -6574.545,E2 -6574.545} C_VEL
LIN {X 0,Y 488.106,Z 396.944,A -85,B 0,C 180,E1 -6575.786,E2 -6575.786} C_VEL
LIN {X 0,Y 488.192,Z 390.87,A -85,B 0,C 180,E1 -6577.238,E2 -6577.238} C_VEL
LIN {X 0,Y 488.454,Z 384.229,A -85,B 0,C 180,E1 -6578.482,E2 -6578.482} C_VEL
LIN {X 0,Y 488.762,Z 375.983,A -85,B 0,C 180,E1 -6579.728,E2 -6579.728} C_VEL
LIN {X 0,Y 489.091,Z 367.529,A -85,B 0,C 180,E1 -6580.767,E2 -6580.767} C_VEL
LIN {X 0,Y 489.54,Z 357.08,A -85,B 0,C 180,E1 -6581.806,E2 -6581.806} C_VEL
LIN {X 0,Y 489.9,Z 345.834,A -85,B 0,C 180,E1 -6582.705,E2 -6582.705} C_VEL
LIN {X 0,Y 490.268,Z 335.386,A -85,B 0,C 180,E1 -6583.366,E2 -6583.366} C_VEL
LIN {X 0,Y 490.681,Z 323.736,A -85,B 0,C 180,E1 -6583.935,E2 -6583.935} C_VEL
LIN {X 0,Y 490.687,Z 313.483,A -85,B 0,C 180,E1 -6584.318,E2 -6584.318} C_VEL
LIN {X 0,Y 488.495,Z 300.518,A -85,B 0,C 180,E1 -6584.708,E2 -6584.708} C_VEL
LIN {X 0,Y 488.383,Z 299.527,A -85,B 0,C 180,E1 -6584.747,E2 -6584.747} C_VEL
LIN {X 0,Y 488.623,Z 289.612,A -85,B 0,C 180,E1 -6587.956,E2 -6587.956} C_VEL
LIN {X 0,Y 488.863,Z 280.031,A -85,B 0,C 180,E1 -6591.065,E2 -6591.065} C_VEL
LIN {X 0,Y 489.092,Z 270.362,A -85,B 0,C 180,E1 -6594.176,E2 -6594.176} C_VEL
LIN {X 0,Y 489.457,Z 260.896,A -85,B 0,C 180,E1 -6597.355,E2 -6597.355} C_VEL
LIN {X 0,Y 489.747,Z 251.618,A -85,B 0,C 180,E1 -6600.569,E2 -6600.569} C_VEL
LIN {X 0,Y 490.11,Z 242.849,A -85,B 0,C 180,E1 -6603.726,E2 -6603.726} C_VEL
LIN {X 0,Y 490.242,Z 236.756,A -85,B 0,C 180,E1 -6606,E2 -6606} C_VEL
LIN {X 0,Y 489.207,Z 230.291,A -85,B 0,C 180,E1 -6608.613,E2 -6608.613} C_VEL
LIN {X 0,Y 488.726,Z 227.61,A -85,B 0,C 180,E1 -6609.787,E2 -6609.787} C_VEL
LIN {X 0,Y 488.715,Z 227.61,A -85,B 0,C 180,E1 -6612.827,E2 -6612.827} C_VEL
LIN {X 0,Y 488.707,Z 227.614,A -85,B 0,C 180,E1 -6615.977,E2 -6615.977} C_VEL
LIN {X 0,Y 488.714,Z 227.608,A -85,B 0,C 180,E1 -6618.585,E2 -6618.585} C_VEL
LIN {X 0,Y 488.707,Z 227.613,A -85,B 0,C 180,E1 -6620.948,E2 -6620.948} C_VEL
LIN {X 0,Y 488.671,Z 227.611,A -85,B 0,C 180,E1 -6623.867,E2 -6623.867} C_VEL
LIN {X 0,Y 488.704,Z 227.609,A -85,B 0,C 180,E1 -6626.874,E2 -6626.874} C_VEL
LIN {X 0,Y 488.726,Z 227.607,A -85,B 0,C 180,E1 -6629.781,E2 -6629.781} C_VEL
LIN {X 0,Y 488.732,Z 227.607,A -85,B 0,C 180,E1 -6633.072,E2 -6633.072} C_VEL
LIN {X 0,Y 488.718,Z 227.609,A -85,B 0,C 180,E1 -6635.353,E2 -6635.353} C_VEL
LIN {X 0,Y 488.705,Z 227.609,A -85,B 0,C 180,E1 -6638.044,E2 -6638.044} C_VEL
LIN {X 0,Y 488.742,Z 227.606,A -85,B 0,C 180,E1 -6640.687,E2 -6640.687} C_VEL
LIN {X 0,Y 488.715,Z 227.612,A -85,B 0,C 180,E1 -6644.143,E2 -6644.143} C_VEL
LIN {X 0,Y 488.713,Z 227.606,A -85,B 0,C 180,E1 -6646.698,E2 -6646.698} C_VEL
LIN {X 0,Y 488.704,Z 227.61,A -85,B 0,C 180,E1 -6649.225,E2 -6649.225} C_VEL
LIN {X 0,Y 488.876,Z 227.589,A -85,B 0,C 180,E1 -6652.724,E2 -6652.724} C_VEL
LIN {X 0,Y 488.813,Z 227.598,A -85,B 0,C 180,E1 -6655.051,E2 -6655.051} C_VEL
LIN {X 0,Y 488.967,Z 227.576,A -85,B 0,C 180,E1 -6657.529,E2 -6657.529} C_VEL
LIN {X 0,Y 488.976,Z 227.579,A -85,B 0,C 180,E1 -6660,E2 -6660} C_VEL
LIN {X 0,Y 488.958,Z 227.577,A -85,B 0,C 180,E1 -6662.471,E2 -6662.471} C_VEL
LIN {X 0,Y 488.809,Z 227.596,A -85,B 0,C 180,E1 -6665.776,E2 -6665.776} C_VEL
LIN {X 0,Y 488.767,Z 227.599,A -85,B 0,C 180,E1 -6668.267,E2 -6668.267} C_VEL
LIN {X 0,Y 488.811,Z 227.595,A -85,B 0,C 180,E1 -6671.612,E2 -6671.612} C_VEL
LIN {X 0,Y 488.769,Z 227.601,A -85,B 0,C 180,E1 -6675,E2 -6675} C_VEL
LIN {X 0,Y 488.755,Z 227.604,A -85,B 0,C 180,E1 -6678.442,E2 -6678.442} C_VEL
LIN {X 0,Y 488.714,Z 227.61,A -85,B 0,C 180,E1 -6681.071,E2 -6681.071} C_VEL
LIN {X 0,Y 488.669,Z 227.613,A -85,B 0,C 180,E1 -6683.747,E2 -6683.747} C_VEL
LIN {X 0,Y 488.673,Z 227.614,A -85,B 0,C 180,E1 -6686.477,E2 -6686.477} C_VEL
LIN {X 0,Y 488.707,Z 227.607,A -85,B 0,C 180,E1 -6689.272,E2 -6689.272} C_VEL
LIN {X 0,Y 488.71,Z 227.612,A -85,B 0,C 180,E1 -6692.147,E2 -6692.147} C_VEL
LIN {X 0,Y 488.721,Z 227.608,A -85,B 0,C 180,E1 -6695.115,E2 -6695.115} C_VEL
LIN {X 0,Y 488.684,Z 227.612,A -85,B 0,C 180,E1 -6698.2,E2 -6698.2} C_VEL
LIN {X 0,Y 488.726,Z 227.607,A -85,B 0,C 180,E1 -6700.344,E2 -6700.344} C_VEL
LIN {X 0,Y 488.684,Z 227.611,A -85,B 0,C 180,E1 -6703.655,E2 -6703.655} C_VEL
LIN {X 0,Y 488.671,Z 227.616,A -85,B 0,C 180,E1 -6706.342,E2 -6706.342} C_VEL
LIN {X 0,Y 488.673,Z 227.615,A -85,B 0,C 180,E1 -6709.669,E2 -6709.669} C_VEL
LIN {X 0,Y 488.676,Z 227.612,A -85,B 0,C 180,E1 -6712.279,E2 -6712.279} C_VEL
LIN {X 0,Y 488.726,Z 227.608,A -85,B 0,C 180,E1 -6715.053,E2 -6715.053} C_VEL
LIN {X 0,Y 488.666,Z 227.615,A -85,B 0,C 180,E1 -6718.054,E2 -6718.054} C_VEL
LIN {X 0,Y 488.414,Z 227.648,A -85,B 0,C 180,E1 -6720.708,E2 -6720.708} C_VEL
LIN {X 0,Y 488.326,Z 227.775,A -85,B 0,C 180,E1 -6721.644,E2 -6721.644} C_VEL
LIN {X 0,Y 488.226,Z 230.52,A -85,B 0,C 180,E1 -6724.255,E2 -6724.255} C_VEL
LIN {X 0,Y 487.562,Z 231.312,A -85,B 0,C 180,E1 -6724.937,E2 -6724.937} C_VEL
LIN {X 0,Y 484.688,Z 232.77,A -85,B 0,C 180,E1 -6726.042,E2 -6726.042} C_VEL
LIN {X 0,Y 482.243,Z 233.951,A -85,B 0,C 180,E1 -6726.932,E2 -6726.932} C_VEL
LIN {X 0,Y 481.179,Z 234.774,A -85,B 0,C 180,E1 -6727.621,E2 -6727.621} C_VEL
LIN {X 0,Y 481.086,Z 235.03,A -85,B 0,C 180,E1 -6727.855,E2 -6727.855} C_VEL
LIN {X 0,Y 481.079,Z 237.7,A -85,B 0,C 180,E1 -6730.365,E2 -6730.365} C_VEL
LIN {X 0,Y 481.055,Z 240.568,A -85,B 0,C 180,E1 -6733.01,E2 -6733.01} C_VEL
LIN {X 0,Y 481.053,Z 243.473,A -85,B 0,C 180,E1 -6735.618,E2 -6735.618} C_VEL
LIN {X 0,Y 481.066,Z 247.422,A -85,B 0,C 180,E1 -6739.051,E2 -6739.051} C_VEL
LIN {X 0,Y 481.063,Z 247.674,A -85,B 0,C 180,E1 -6739.184,E2 -6739.184} C_VEL
LIN {X 0,Y 484.073,Z 261.296,A -85,B 0,C 180,E1 -6739.675,E2 -6739.675} C_VEL
LIN {X 0,Y 483.855,Z 274.079,A -85,B 0,C 180,E1 -6740.225,E2 -6740.225} C_VEL
LIN {X 0,Y 483.464,Z 285.732,A -85,B 0,C 180,E1 -6740.903,E2 -6740.903} C_VEL
LIN {X 0,Y 482.956,Z 297.047,A -85,B 0,C 180,E1 -6741.744,E2 -6741.744} C_VEL
LIN {X 0,Y 482.641,Z 307.059,A -85,B 0,C 180,E1 -6742.679,E2 -6742.679} C_VEL
LIN {X 0,Y 482.257,Z 316.152,A -85,B 0,C 180,E1 -6743.724,E2 -6743.724} C_VEL
LIN {X 0,Y 481.805,Z 324.997,A -85,B 0,C 180,E1 -6744.978,E2 -6744.978} C_VEL
LIN {X 0,Y 481.464,Z 332.124,A -85,B 0,C 180,E1 -6746.232,E2 -6746.232} C_VEL
LIN {X 0,Y 481.082,Z 337.84,A -85,B 0,C 180,E1 -6747.487,E2 -6747.487} C_VEL
LIN {X 0,Y 481.064,Z 342.321,A -85,B 0,C 180,E1 -6748.743,E2 -6748.743} C_VEL
LIN {X 0,Y 480.846,Z 345.755,A -85,B 0,C 180,E1 -6749.999,E2 -6749.999} C_VEL
LIN {X 0,Y 480.803,Z 347.475,A -85,B 0,C 180,E1 -6750.836,E2 -6750.836} C_VEL
LIN {X 0,Y 480.938,Z 349.695,A -85,B 0,C 180,E1 -6752.511,E2 -6752.511} C_VEL
LIN {X 0,Y 480.947,Z 350.237,A -85,B 0,C 180,E1 -6753.35,E2 -6753.35} C_VEL
LIN {X 0,Y 480.923,Z 350.356,A -85,B 0,C 180,E1 -6754.189,E2 -6754.189} C_VEL
LIN {X 0,Y 480.936,Z 349.435,A -85,B 0,C 180,E1 -6755.87,E2 -6755.87} C_VEL
LIN {X 0,Y 480.948,Z 348.4,A -85,B 0,C 180,E1 -6756.712,E2 -6756.712} C_VEL
LIN {X 0,Y 480.975,Z 346.917,A -85,B 0,C 180,E1 -6757.555,E2 -6757.555} C_VEL
LIN {X 0,Y 481.047,Z 343.909,A -85,B 0,C 180,E1 -6758.823,E2 -6758.823} C_VEL
LIN {X 0,Y 481.152,Z 339.842,A -85,B 0,C 180,E1 -6760.094,E2 -6760.094} C_VEL
LIN {X 0,Y 481.422,Z 333.585,A -85,B 0,C 180,E1 -6761.578,E2 -6761.578} C_VEL
LIN {X 0,Y 481.749,Z 326.747,A -85,B 0,C 180,E1 -6762.853,E2 -6762.853} C_VEL
LIN {X 0,Y 482.044,Z 319.739,A -85,B 0,C 180,E1 -6763.918,E2 -6763.918} C_VEL
LIN {X 0,Y 482.444,Z 311.254,A -85,B 0,C 180,E1 -6764.984,E2 -6764.984} C_VEL
LIN {X 0,Y 482.932,Z 300.719,A -85,B 0,C 180,E1 -6766.05,E2 -6766.05} C_VEL
LIN {X 0,Y 483.331,Z 290.242,A -85,B 0,C 180,E1 -6766.905,E2 -6766.905} C_VEL
LIN {X 0,Y 483.727,Z 278.664,A -85,B 0,C 180,E1 -6767.654,E2 -6767.654} C_VEL
LIN {X 0,Y 484.045,Z 266.016,A -85,B 0,C 180,E1 -6768.266,E2 -6768.266} C_VEL
LIN {X 0,Y 484.011,Z 260.169,A -85,B 0,C 180,E1 -6768.493,E2 -6768.493} C_VEL
LIN {X 0,Y 481.002,Z 247.622,A -85,B 0,C 180,E1 -6768.97,E2 -6768.97} C_VEL
LIN {X 0,Y 480.986,Z 243.833,A -85,B 0,C 180,E1 -6772.326,E2 -6772.326} C_VEL
LIN {X 0,Y 481.119,Z 240.795,A -85,B 0,C 180,E1 -6775.085,E2 -6775.085} C_VEL
LIN {X 0,Y 481.123,Z 237.845,A -85,B 0,C 180,E1 -6777.867,E2 -6777.867} C_VEL
LIN {X 0,Y 481.169,Z 234.839,A -85,B 0,C 180,E1 -6780.743,E2 -6780.743} C_VEL
LIN {X 0,Y 481.238,Z 231.807,A -85,B 0,C 180,E1 -6783.706,E2 -6783.706} C_VEL
LIN {X 0,Y 481.309,Z 228.901,A -85,B 0,C 180,E1 -6786.572,E2 -6786.572} C_VEL
LIN {X 0,Y 481.547,Z 228.504,A -85,B 0,C 180,E1 -6788.869,E2 -6788.869} C_VEL
LIN {X 0,Y 481.642,Z 228.488,A -85,B 0,C 180,E1 -6791.911,E2 -6791.911} C_VEL
LIN {X 0,Y 481.653,Z 228.492,A -85,B 0,C 180,E1 -6794.456,E2 -6794.456} C_VEL
LIN {X 0,Y 481.635,Z 228.493,A -85,B 0,C 180,E1 -6797.838,E2 -6797.838} C_VEL
LIN {X 0,Y 481.652,Z 228.49,A -85,B 0,C 180,E1 -6800.653,E2 -6800.653} C_VEL
LIN {X 0,Y 481.624,Z 228.489,A -85,B 0,C 180,E1 -6803.374,E2 -6803.374} C_VEL
LIN {X 0,Y 481.684,Z 228.483,A -85,B 0,C 180,E1 -6806.328,E2 -6806.328} C_VEL
LIN {X 0,Y 481.64,Z 228.491,A -85,B 0,C 180,E1 -6809.417,E2 -6809.417} C_VEL
LIN {X 0,Y 481.692,Z 228.484,A -85,B 0,C 180,E1 -6812.167,E2 -6812.167} C_VEL
LIN {X 0,Y 481.709,Z 228.479,A -85,B 0,C 180,E1 -6814.969,E2 -6814.969} C_VEL
LIN {X 0,Y 481.639,Z 228.491,A -85,B 0,C 180,E1 -6817.704,E2 -6817.704} C_VEL
LIN {X 0,Y 481.694,Z 228.483,A -85,B 0,C 180,E1 -6820.392,E2 -6820.392} C_VEL
LIN {X 0,Y 481.678,Z 228.484,A -85,B 0,C 180,E1 -6823.033,E2 -6823.033} C_VEL
LIN {X 0,Y 481.68,Z 228.488,A -85,B 0,C 180,E1 -6825.638,E2 -6825.638} C_VEL
LIN {X 0,Y 481.739,Z 228.475,A -85,B 0,C 180,E1 -6828.215,E2 -6828.215} C_VEL
LIN {X 0,Y 481.749,Z 228.475,A -85,B 0,C 180,E1 -6831.611,E2 -6831.611} C_VEL
LIN {X 0,Y 481.822,Z 228.469,A -85,B 0,C 180,E1 -6834.14,E2 -6834.14} C_VEL
LIN {X 0,Y 481.917,Z 228.456,A -85,B 0,C 180,E1 -6837.492,E2 -6837.492} C_VEL
LIN {X 0,Y 481.872,Z 228.462,A -85,B 0,C 180,E1 -6840.836,E2 -6840.836} C_VEL
LIN {X 0,Y 481.917,Z 228.455,A -85,B 0,C 180,E1 -6842.507,E2 -6842.507} C_VEL
LIN {X 0,Y 481.818,Z 228.467,A -85,B 0,C 180,E1 -6845.86,E2 -6845.86} C_VEL
LIN {X 0,Y 481.751,Z 228.477,A -85,B 0,C 180,E1 -6848.388,E2 -6848.388} C_VEL
LIN {X 0,Y 481.738,Z 228.479,A -85,B 0,C 180,E1 -6851.785,E2 -6851.785} C_VEL
LIN {X 0,Y 481.731,Z 228.479,A -85,B 0,C 180,E1 -6855.225,E2 -6855.225} C_VEL
LIN {X 0,Y 481.701,Z 228.482,A -85,B 0,C 180,E1 -6858.722,E2 -6858.722} C_VEL
LIN {X 0,Y 481.634,Z 228.49,A -85,B 0,C 180,E1 -6861.395,E2 -6861.395} C_VEL
LIN {X 0,Y 481.658,Z 228.486,A -85,B 0,C 180,E1 -6864.114,E2 -6864.114} C_VEL
LIN {X 0,Y 481.742,Z 228.478,A -85,B 0,C 180,E1 -6867.141,E2 -6867.141} C_VEL
LIN {X 0,Y 481.678,Z 228.485,A -85,B 0,C 180,E1 -6869.741,E2 -6869.741} C_VEL
LIN {X 0,Y 481.662,Z 228.486,A -85,B 0,C 180,E1 -6872.675,E2 -6872.675} C_VEL
LIN {X 0,Y 481.627,Z 228.49,A -85,B 0,C 180,E1 -6875.71,E2 -6875.71} C_VEL
LIN {X 0,Y 481.663,Z 228.486,A -85,B 0,C 180,E1 -6878.86,E2 -6878.86} C_VEL
LIN {X 0,Y 481.643,Z 228.491,A -85,B 0,C 180,E1 -6881.914,E2 -6881.914} C_VEL
LIN {X 0,Y 481.651,Z 228.489,A -85,B 0,C 180,E1 -6884.459,E2 -6884.459} C_VEL
LIN {X 0,Y 481.642,Z 228.492,A -85,B 0,C 180,E1 -6887.841,E2 -6887.841} C_VEL
LIN {X 0,Y 481.735,Z 228.598,A -85,B 0,C 180,E1 -6889.871,E2 -6889.871} C_VEL
LIN {X 0,Y 483.026,Z 236.147,A -85,B 0,C 180,E1 -6893.154,E2 -6893.154} C_VEL
LIN {X 0,Y 483.283,Z 239.55,A -85,B 0,C 180,E1 -6894.525,E2 -6894.525} C_VEL
LIN {X 0,Y 482.945,Z 247.613,A -85,B 0,C 180,E1 -6897.569,E2 -6897.569} C_VEL
LIN {X 0,Y 482.664,Z 253.918,A -85,B 0,C 180,E1 -6899.846,E2 -6899.846} C_VEL
LIN {X 0,Y 482.33,Z 263.353,A -85,B 0,C 180,E1 -6903.149,E2 -6903.149} C_VEL
LIN {X 0,Y 481.975,Z 272.808,A -85,B 0,C 180,E1 -6906.362,E2 -6906.362} C_VEL
LIN {X 0,Y 481.769,Z 282.478,A -85,B 0,C 180,E1 -6909.507,E2 -6909.507} C_VEL
LIN {X 0,Y 481.547,Z 290.716,A -85,B 0,C 180,E1 -6912.154,E2 -6912.154} C_VEL
LIN {X 0,Y 481.33,Z 299.617,A -85,B 0,C 180,E1 -6915.052,E2 -6915.052} C_VEL
LIN {X 0,Y 483.611,Z 313.141,A -85,B 0,C 180,E1 -6915.457,E2 -6915.457} C_VEL
LIN {X 0,Y 483.962,Z 317.017,A -85,B 0,C 180,E1 -6915.602,E2 -6915.602} C_VEL
LIN {X 0,Y 483.572,Z 329.516,A -85,B 0,C 180,E1 -6916.126,E2 -6916.126} C_VEL
LIN {X 0,Y 483.168,Z 340.958,A -85,B 0,C 180,E1 -6916.779,E2 -6916.779} C_VEL
LIN {X 0,Y 482.759,Z 352.21,A -85,B 0,C 180,E1 -6917.602,E2 -6917.602} C_VEL
LIN {X 0,Y 482.353,Z 362.619,A -85,B 0,C 180,E1 -6918.551,E2 -6918.551} C_VEL
LIN {X 0,Y 481.955,Z 371.124,A -85,B 0,C 180,E1 -6919.499,E2 -6919.499} C_VEL
LIN {X 0,Y 481.635,Z 378.969,A -85,B 0,C 180,E1 -6920.553,E2 -6920.553} C_VEL
LIN {X 0,Y 481.323,Z 386.628,A -85,B 0,C 180,E1 -6921.817,E2 -6921.817} C_VEL
LIN {X 0,Y 481.058,Z 393.685,A -85,B 0,C 180,E1 -6923.289,E2 -6923.289} C_VEL
LIN {X 0,Y 480.998,Z 398.377,A -85,B 0,C 180,E1 -6924.551,E2 -6924.551} C_VEL
LIN {X 0,Y 480.846,Z 401.961,A -85,B 0,C 180,E1 -6925.81,E2 -6925.81} C_VEL
LIN {X 0,Y 480.891,Z 403.809,A -85,B 0,C 180,E1 -6926.65,E2 -6926.65} C_VEL
LIN {X 0,Y 480.789,Z 406.184,A -85,B 0,C 180,E1 -6928.326,E2 -6928.326} C_VEL
LIN {X 0,Y 480.742,Z 407,A -85,B 0,C 180,E1 -6930.001,E2 -6930.001} C_VEL
LIN {X 0,Y 480.79,Z 406.183,A -85,B 0,C 180,E1 -6931.677,E2 -6931.677} C_VEL
LIN {X 0,Y 480.892,Z 403.808,A -85,B 0,C 180,E1 -6933.353,E2 -6933.353} C_VEL
LIN {X 0,Y 480.854,Z 400.892,A -85,B 0,C 180,E1 -6934.612,E2 -6934.612} C_VEL
LIN {X 0,Y 481.024,Z 396.944,A -85,B 0,C 180,E1 -6935.871,E2 -6935.871} C_VEL
LIN {X 0,Y 481.117,Z 390.87,A -85,B 0,C 180,E1 -6937.345,E2 -6937.345} C_VEL
LIN {X 0,Y 481.427,Z 384.229,A -85,B 0,C 180,E1 -6938.607,E2 -6938.607} C_VEL
LIN {X 0,Y 481.754,Z 375.984,A -85,B 0,C 180,E1 -6939.871,E2 -6939.871} C_VEL
LIN {X 0,Y 482.109,Z 367.529,A -85,B 0,C 180,E1 -6940.925,E2 -6940.925} C_VEL
LIN {X 0,Y 482.567,Z 357.079,A -85,B 0,C 180,E1 -6941.979,E2 -6941.979} C_VEL
LIN {X 0,Y 482.97,Z 345.862,A -85,B 0,C 180,E1 -6942.888,E2 -6942.888} C_VEL
LIN {X 0,Y 483.353,Z 335.385,A -85,B 0,C 180,E1 -6943.561,E2 -6943.561} C_VEL
LIN {X 0,Y 483.789,Z 323.736,A -85,B 0,C 180,E1 -6944.138,E2 -6944.138} C_VEL
LIN {X 0,Y 483.851,Z 314.651,A -85,B 0,C 180,E1 -6944.485,E2 -6944.485} C_VEL
LIN {X 0,Y 481.661,Z 301.542,A -85,B 0,C 180,E1 -6944.903,E2 -6944.903} C_VEL
LIN {X 0,Y 481.325,Z 299.527,A -85,B 0,C 180,E1 -6944.968,E2 -6944.968} C_VEL
LIN {X 0,Y 481.558,Z 290.71,A -85,B 0,C 180,E1 -6947.848,E2 -6947.848} C_VEL
LIN {X 0,Y 481.799,Z 280.917,A -85,B 0,C 180,E1 -6951.002,E2 -6951.002} C_VEL
LIN {X 0,Y 482.027,Z 271.438,A -85,B 0,C 180,E1 -6954.096,E2 -6954.096} C_VEL
LIN {X 0,Y 482.434,Z 262.075,A -85,B 0,C 180,E1 -6957.297,E2 -6957.297} C_VEL
LIN {X 0,Y 482.807,Z 251.136,A -85,B 0,C 180,E1 -6961.157,E2 -6961.157} C_VEL
LIN {X 0,Y 483.136,Z 243.431,A -85,B 0,C 180,E1 -6963.988,E2 -6963.988} C_VEL
LIN {X 0,Y 483.267,Z 237.911,A -85,B 0,C 180,E1 -6966.086,E2 -6966.086} C_VEL
LIN {X 0,Y 482.187,Z 231.274,A -85,B 0,C 180,E1 -6968.811,E2 -6968.811} C_VEL
LIN {X 0,Y 481.681,Z 228.488,A -85,B 0,C 180,E1 -6970.071,E2 -6970.071} C_VEL
LIN {X 0,Y 481.645,Z 228.49,A -85,B 0,C 180,E1 -6973.3,E2 -6973.3} C_VEL
LIN {X 0,Y 481.665,Z 228.491,A -85,B 0,C 180,E1 -6975.641,E2 -6975.641} C_VEL
LIN {X 0,Y 481.663,Z 228.488,A -85,B 0,C 180,E1 -6978.959,E2 -6978.959} C_VEL
LIN {X 0,Y 481.655,Z 228.486,A -85,B 0,C 180,E1 -6981.994,E2 -6981.994} C_VEL
LIN {X 0,Y 481.686,Z 228.481,A -85,B 0,C 180,E1 -6985.318,E2 -6985.318} C_VEL
LIN {X 0,Y 481.641,Z 228.494,A -85,B 0,C 180,E1 -6988.311,E2 -6988.311} C_VEL
LIN {X 0,Y 481.681,Z 228.485,A -85,B 0,C 180,E1 -6991.217,E2 -6991.217} C_VEL
LIN {X 0,Y 481.677,Z 228.486,A -85,B 0,C 180,E1 -6994.041,E2 -6994.041} C_VEL
LIN {X 0,Y 481.681,Z 228.487,A -85,B 0,C 180,E1 -6996.812,E2 -6996.812} C_VEL
LIN {X 0,Y 481.702,Z 228.482,A -85,B 0,C 180,E1 -6999.503,E2 -6999.503} C_VEL
LIN {X 0,Y 481.677,Z 228.487,A -85,B 0,C 180,E1 -7002.157,E2 -7002.157} C_VEL
LIN {X 0,Y 481.735,Z 228.476,A -85,B 0,C 180,E1 -7004.776,E2 -7004.776} C_VEL
LIN {X 0,Y 481.74,Z 228.476,A -85,B 0,C 180,E1 -7008.215,E2 -7008.215} C_VEL
LIN {X 0,Y 481.738,Z 228.479,A -85,B 0,C 180,E1 -7011.611,E2 -7011.611} C_VEL
LIN {X 0,Y 481.813,Z 228.468,A -85,B 0,C 180,E1 -7014.14,E2 -7014.14} C_VEL
LIN {X 0,Y 481.933,Z 228.453,A -85,B 0,C 180,E1 -7017.493,E2 -7017.493} C_VEL
LIN {X 0,Y 481.947,Z 228.454,A -85,B 0,C 180,E1 -7020,E2 -7020} C_VEL
LIN {X 0,Y 481.924,Z 228.453,A -85,B 0,C 180,E1 -7022.508,E2 -7022.508} C_VEL
LIN {X 0,Y 481.771,Z 228.472,A -85,B 0,C 180,E1 -7025.861,E2 -7025.861} C_VEL
LIN {X 0,Y 481.726,Z 228.477,A -85,B 0,C 180,E1 -7028.389,E2 -7028.389} C_VEL
LIN {X 0,Y 481.757,Z 228.474,A -85,B 0,C 180,E1 -7031.785,E2 -7031.785} C_VEL
LIN {X 0,Y 481.75,Z 228.475,A -85,B 0,C 180,E1 -7035.224,E2 -7035.224} C_VEL
LIN {X 0,Y 481.716,Z 228.48,A -85,B 0,C 180,E1 -7038.722,E2 -7038.722} C_VEL
LIN {X 0,Y 481.653,Z 228.49,A -85,B 0,C 180,E1 -7041.395,E2 -7041.395} C_VEL
LIN {X 0,Y 481.648,Z 228.487,A -85,B 0,C 180,E1 -7044.115,E2 -7044.115} C_VEL
LIN {X 0,Y 481.649,Z 228.488,A -85,B 0,C 180,E1 -7047.114,E2 -7047.114} C_VEL
LIN {X 0,Y 481.673,Z 228.484,A -85,B 0,C 180,E1 -7049.742,E2 -7049.742} C_VEL
LIN {X 0,Y 481.678,Z 228.485,A -85,B 0,C 180,E1 -7052.674,E2 -7052.674} C_VEL
LIN {X 0,Y 481.639,Z 228.491,A -85,B 0,C 180,E1 -7055.71,E2 -7055.71} C_VEL
LIN {X 0,Y 481.676,Z 228.488,A -85,B 0,C 180,E1 -7058.859,E2 -7058.859} C_VEL
LIN {X 0,Y 481.653,Z 228.487,A -85,B 0,C 180,E1 -7061.911,E2 -7061.911} C_VEL
LIN {X 0,Y 481.661,Z 228.49,A -85,B 0,C 180,E1 -7064.458,E2 -7064.458} C_VEL
LIN {X 0,Y 481.618,Z 228.49,A -85,B 0,C 180,E1 -7066.855,E2 -7066.855} C_VEL
LIN {X 0,Y 481.638,Z 228.492,A -85,B 0,C 180,E1 -7070.054,E2 -7070.054} C_VEL
LIN {X 0,Y 481.63,Z 228.49,A -85,B 0,C 180,E1 -7072.201,E2 -7072.201} C_VEL
LIN {X 0,Y 481.69,Z 228.486,A -85,B 0,C 180,E1 -7075.317,E2 -7075.317} C_VEL
LIN {X 0,Y 481.587,Z 228.498,A -85,B 0,C 180,E1 -7078.306,E2 -7078.306} C_VEL
LIN {X 0,Y 481.301,Z 228.535,A -85,B 0,C 180,E1 -7081.191,E2 -7081.191} C_VEL
LIN {X 0,Y 481.21,Z 229.024,A -85,B 0,C 180,E1 -7082.136,E2 -7082.136} C_VEL
LIN {X 0,Y 481.213,Z 231.954,A -85,B 0,C 180,E1 -7084.941,E2 -7084.941} C_VEL
LIN {X 0,Y 481.086,Z 235.03,A -85,B 0,C 180,E1 -7087.855,E2 -7087.855} C_VEL
LIN {X 0,Y 480.391,Z 235.837,A -85,B 0,C 180,E1 -7088.547,E2 -7088.547} C_VEL
LIN {X 0,Y 477.501,Z 237.316,A -85,B 0,C 180,E1 -7089.668,E2 -7089.668} C_VEL
LIN {X 0,Y 475.087,Z 238.508,A -85,B 0,C 180,E1 -7090.572,E2 -7090.572} C_VEL
LIN {X 0,Y 474.079,Z 239.346,A -85,B 0,C 180,E1 -7091.271,E2 -7091.271} C_VEL
LIN {X 0,Y 474.01,Z 239.604,A -85,B 0,C 180,E1 -7091.508,E2 -7091.508} C_VEL
LIN {X 0,Y 474.018,Z 242.898,A -85,B 0,C 180,E1 -7094.52,E2 -7094.52} C_VEL
LIN {X 0,Y 474.012,Z 246.976,A -85,B 0,C 180,E1 -7098.115,E2 -7098.115} C_VEL
LIN {X 0,Y 474.015,Z 247.977,A -85,B 0,C 180,E1 -7098.967,E2 -7098.967} C_VEL
LIN {X 0,Y 476.992,Z 261.282,A -85,B 0,C 180,E1 -7099.453,E2 -7099.453} C_VEL
LIN {X 0,Y 477.069,Z 270.02,A -85,B 0,C 180,E1 -7099.817,E2 -7099.817} C_VEL
LIN {X 0,Y 476.715,Z 281.947,A -85,B 0,C 180,E1 -7100.452,E2 -7100.452} C_VEL
LIN {X 0,Y 476.245,Z 292.753,A -85,B 0,C 180,E1 -7101.192,E2 -7101.192} C_VEL
LIN {X 0,Y 475.837,Z 302.354,A -85,B 0,C 180,E1 -7102.01,E2 -7102.01} C_VEL
LIN {X 0,Y 475.441,Z 311.797,A -85,B 0,C 180,E1 -7102.994,E2 -7102.994} C_VEL
LIN {X 0,Y 475.098,Z 320.12,A -85,B 0,C 180,E1 -7104.055,E2 -7104.055} C_VEL
LIN {X 0,Y 474.593,Z 328.262,A -85,B 0,C 180,E1 -7105.327,E2 -7105.327} C_VEL
LIN {X 0,Y 474.301,Z 333.827,A -85,B 0,C 180,E1 -7106.388,E2 -7106.388} C_VEL
LIN {X 0,Y 474.022,Z 338.469,A -85,B 0,C 180,E1 -7107.449,E2 -7107.449} C_VEL
LIN {X 0,Y 473.999,Z 342.904,A -85,B 0,C 180,E1 -7108.724,E2 -7108.724} C_VEL
LIN {X 0,Y 473.766,Z 346.301,A -85,B 0,C 180,E1 -7109.999,E2 -7109.999} C_VEL
LIN {X 0,Y 473.769,Z 349.273,A -85,B 0,C 180,E1 -7111.699,E2 -7111.699} C_VEL
LIN {X 0,Y 473.878,Z 350.169,A -85,B 0,C 180,E1 -7112.549,E2 -7112.549} C_VEL
LIN {X 0,Y 473.872,Z 350.682,A -85,B 0,C 180,E1 -7113.4,E2 -7113.4} C_VEL
LIN {X 0,Y 473.783,Z 350.487,A -85,B 0,C 180,E1 -7115.105,E2 -7115.105} C_VEL
LIN {X 0,Y 473.867,Z 349.248,A -85,B 0,C 180,E1 -7116.438,E2 -7116.438} C_VEL
LIN {X 0,Y 473.915,Z 347.236,A -85,B 0,C 180,E1 -7117.669,E2 -7117.669} C_VEL
LIN {X 0,Y 473.993,Z 344.186,A -85,B 0,C 180,E1 -7118.955,E2 -7118.955} C_VEL
LIN {X 0,Y 474.112,Z 340.076,A -85,B 0,C 180,E1 -7120.245,E2 -7120.245} C_VEL
LIN {X 0,Y 474.414,Z 333.772,A -85,B 0,C 180,E1 -7121.752,E2 -7121.752} C_VEL
LIN {X 0,Y 474.761,Z 326.88,A -85,B 0,C 180,E1 -7123.046,E2 -7123.046} C_VEL
LIN {X 0,Y 475.179,Z 318.197,A -85,B 0,C 180,E1 -7124.342,E2 -7124.342} C_VEL
LIN {X 0,Y 475.604,Z 309.27,A -85,B 0,C 180,E1 -7125.424,E2 -7125.424} C_VEL
LIN {X 0,Y 476.072,Z 299.541,A -85,B 0,C 180,E1 -7126.387,E2 -7126.387} C_VEL
LIN {X 0,Y 476.527,Z 288.49,A -85,B 0,C 180,E1 -7127.265,E2 -7127.265} C_VEL
LIN {X 0,Y 476.965,Z 276.175,A -85,B 0,C 180,E1 -7128.024,E2 -7128.024} C_VEL
LIN {X 0,Y 477.302,Z 264.586,A -85,B 0,C 180,E1 -7128.561,E2 -7128.561} C_VEL
LIN {X 0,Y 477.041,Z 260.909,A -85,B 0,C 180,E1 -7128.71,E2 -7128.71} C_VEL
LIN {X 0,Y 473.937,Z 248.035,A -85,B 0,C 180,E1 -7129.208,E2 -7129.208} C_VEL
LIN {X 0,Y 473.894,Z 245.155,A -85,B 0,C 180,E1 -7131.761,E2 -7131.761} C_VEL
LIN {X 0,Y 474.003,Z 242.124,A -85,B 0,C 180,E1 -7134.527,E2 -7134.527} C_VEL
LIN {X 0,Y 474.066,Z 239.106,A -85,B 0,C 180,E1 -7137.358,E2 -7137.358} C_VEL
LIN {X 0,Y 474.105,Z 236.074,A -85,B 0,C 180,E1 -7140.264,E2 -7140.264} C_VEL
LIN {X 0,Y 474.168,Z 233.044,A -85,B 0,C 180,E1 -7143.256,E2 -7143.256} C_VEL
LIN {X 0,Y 474.241,Z 229.919,A -85,B 0,C 180,E1 -7146.353,E2 -7146.353} C_VEL
LIN {X 0,Y 474.265,Z 229.426,A -85,B 0,C 180,E1 -7146.849,E2 -7146.849} C_VEL
LIN {X 0,Y 474.548,Z 229.374,A -85,B 0,C 180,E1 -7149.635,E2 -7149.635} C_VEL
LIN {X 0,Y 474.617,Z 229.364,A -85,B 0,C 180,E1 -7152.235,E2 -7152.235} C_VEL
LIN {X 0,Y 474.614,Z 229.364,A -85,B 0,C 180,E1 -7155.296,E2 -7155.296} C_VEL
LIN {X 0,Y 474.607,Z 229.365,A -85,B 0,C 180,E1 -7158.213,E2 -7158.213} C_VEL
LIN {X 0,Y 474.604,Z 229.365,A -85,B 0,C 180,E1 -7161.542,E2 -7161.542} C_VEL
LIN {X 0,Y 474.62,Z 229.364,A -85,B 0,C 180,E1 -7164.725,E2 -7164.725} C_VEL
LIN {X 0,Y 474.625,Z 229.365,A -85,B 0,C 180,E1 -7167.787,E2 -7167.787} C_VEL
LIN {X 0,Y 474.615,Z 229.368,A -85,B 0,C 180,E1 -7170.884,E2 -7170.884} C_VEL
LIN {X 0,Y 474.657,Z 229.358,A -85,B 0,C 180,E1 -7173.628,E2 -7173.628} C_VEL
LIN {X 0,Y 474.625,Z 229.362,A -85,B 0,C 180,E1 -7176.64,E2 -7176.64} C_VEL
LIN {X 0,Y 474.643,Z 229.36,A -85,B 0,C 180,E1 -7180.089,E2 -7180.089} C_VEL
LIN {X 0,Y 474.637,Z 229.362,A -85,B 0,C 180,E1 -7182.774,E2 -7182.774} C_VEL
LIN {X 0,Y 474.638,Z 229.364,A -85,B 0,C 180,E1 -7185.42,E2 -7185.42} C_VEL
LIN {X 0,Y 474.693,Z 229.353,A -85,B 0,C 180,E1 -7188.037,E2 -7188.037} C_VEL
LIN {X 0,Y 474.714,Z 229.351,A -85,B 0,C 180,E1 -7191.486,E2 -7191.486} C_VEL
LIN {X 0,Y 474.782,Z 229.347,A -85,B 0,C 180,E1 -7194.052,E2 -7194.052} C_VEL
LIN {X 0,Y 474.883,Z 229.332,A -85,B 0,C 180,E1 -7197.455,E2 -7197.455} C_VEL
LIN {X 0,Y 474.896,Z 229.329,A -85,B 0,C 180,E1 -7200,E2 -7200} C_VEL
LIN {X 0,Y 474.883,Z 229.331,A -85,B 0,C 180,E1 -7202.545,E2 -7202.545} C_VEL
LIN {X 0,Y 474.779,Z 229.343,A -85,B 0,C 180,E1 -7205.948,E2 -7205.948} C_VEL
LIN {X 0,Y 474.716,Z 229.354,A -85,B 0,C 180,E1 -7208.514,E2 -7208.514} C_VEL
LIN {X 0,Y 474.692,Z 229.358,A -85,B 0,C 180,E1 -7211.963,E2 -7211.963} C_VEL
LIN {X 0,Y 474.688,Z 229.355,A -85,B 0,C 180,E1 -7215.456,E2 -7215.456} C_VEL
LIN {X 0,Y 474.654,Z 229.358,A -85,B 0,C 180,E1 -7219.011,E2 -7219.011} C_VEL
LIN {X 0,Y 474.577,Z 229.372,A -85,B 0,C 180,E1 -7221.729,E2 -7221.729} C_VEL
LIN {X 0,Y 474.643,Z 229.36,A -85,B 0,C 180,E1 -7224.494,E2 -7224.494} C_VEL
LIN {X 0,Y 474.689,Z 229.355,A -85,B 0,C 180,E1 -7227.339,E2 -7227.339} C_VEL
LIN {X 0,Y 474.599,Z 229.366,A -85,B 0,C 180,E1 -7230.812,E2 -7230.812} C_VEL
LIN {X 0,Y 474.627,Z 229.363,A -85,B 0,C 180,E1 -7233.985,E2 -7233.985} C_VEL
LIN {X 0,Y 474.562,Z 229.372,A -85,B 0,C 180,E1 -7236.9,E2 -7236.9} C_VEL
LIN {X 0,Y 474.619,Z 229.364,A -85,B 0,C 180,E1 -7239.649,E2 -7239.649} C_VEL
LIN {X 0,Y 474.594,Z 229.367,A -85,B 0,C 180,E1 -7242.235,E2 -7242.235} C_VEL
LIN {X 0,Y 474.613,Z 229.367,A -85,B 0,C 180,E1 -7245.298,E2 -7245.298} C_VEL
LIN {X 0,Y 474.617,Z 229.368,A -85,B 0,C 180,E1 -7248.216,E2 -7248.216} C_VEL
LIN {X 0,Y 474.652,Z 229.461,A -85,B 0,C 180,E1 -7249.54,E2 -7249.54} C_VEL
LIN {X 0,Y 475.915,Z 236.625,A -85,B 0,C 180,E1 -7252.74,E2 -7252.74} C_VEL
LIN {X 0,Y 476.309,Z 240.254,A -85,B 0,C 180,E1 -7254.246,E2 -7254.246} C_VEL
LIN {X 0,Y 476.043,Z 247.065,A -85,B 0,C 180,E1 -7256.892,E2 -7256.892} C_VEL
LIN {X 0,Y 475.653,Z 255.05,A -85,B 0,C 180,E1 -7259.845,E2 -7259.845} C_VEL
LIN {X 0,Y 475.295,Z 264.479,A -85,B 0,C 180,E1 -7263.194,E2 -7263.194} C_VEL
LIN {X 0,Y 474.916,Z 273.874,A -85,B 0,C 180,E1 -7266.451,E2 -7266.451} C_VEL
LIN {X 0,Y 474.707,Z 282.165,A -85,B 0,C 180,E1 -7269.189,E2 -7269.189} C_VEL
LIN {X 0,Y 474.459,Z 291.778,A -85,B 0,C 180,E1 -7272.324,E2 -7272.324} C_VEL
LIN {X 0,Y 474.281,Z 299.532,A -85,B 0,C 180,E1 -7274.825,E2 -7274.825} C_VEL
LIN {X 0,Y 476.538,Z 312.685,A -85,B 0,C 180,E1 -7275.222,E2 -7275.222} C_VEL
LIN {X 0,Y 477.072,Z 317.779,A -85,B 0,C 180,E1 -7275.416,E2 -7275.416} C_VEL
LIN {X 0,Y 476.63,Z 330.534,A -85,B 0,C 180,E1 -7275.975,E2 -7275.975} C_VEL
LIN {X 0,Y 476.17,Z 342.696,A -85,B 0,C 180,E1 -7276.701,E2 -7276.701} C_VEL
LIN {X 0,Y 475.759,Z 353.66,A -85,B 0,C 180,E1 -7277.538,E2 -7277.538} C_VEL
LIN {X 0,Y 475.337,Z 363.658,A -85,B 0,C 180,E1 -7278.488,E2 -7278.488} C_VEL
LIN {X 0,Y 474.884,Z 372.796,A -85,B 0,C 180,E1 -7279.556,E2 -7279.556} C_VEL
LIN {X 0,Y 474.481,Z 381.696,A -85,B 0,C 180,E1 -7280.839,E2 -7280.839} C_VEL
LIN {X 0,Y 474.151,Z 388.855,A -85,B 0,C 180,E1 -7282.121,E2 -7282.121} C_VEL
LIN {X 0,Y 473.971,Z 394.743,A -85,B 0,C 180,E1 -7283.45,E2 -7283.45} C_VEL
LIN {X 0,Y 473.845,Z 399.68,A -85,B 0,C 180,E1 -7284.896,E2 -7284.896} C_VEL
LIN {X 0,Y 473.751,Z 401.961,A -85,B 0,C 180,E1 -7285.748,E2 -7285.748} C_VEL
LIN {X 0,Y 473.799,Z 403.809,A -85,B 0,C 180,E1 -7286.6,E2 -7286.6} C_VEL
LIN {X 0,Y 473.695,Z 406.183,A -85,B 0,C 180,E1 -7288.301,E2 -7288.301} C_VEL
LIN {X 0,Y 473.688,Z 406.786,A -85,B 0,C 180,E1 -7289.151,E2 -7289.151} C_VEL
LIN {X 0,Y 473.669,Z 407,A -85,B 0,C 180,E1 -7290.001,E2 -7290.001} C_VEL
LIN {X 0,Y 473.688,Z 406.785,A -85,B 0,C 180,E1 -7290.851,E2 -7290.851} C_VEL
LIN {X 0,Y 473.724,Z 405.194,A -85,B 0,C 180,E1 -7292.552,E2 -7292.552} C_VEL
LIN {X 0,Y 473.8,Z 403.808,A -85,B 0,C 180,E1 -7293.403,E2 -7293.403} C_VEL
LIN {X 0,Y 473.776,Z 400.892,A -85,B 0,C 180,E1 -7294.681,E2 -7294.681} C_VEL
LIN {X 0,Y 473.943,Z 396.944,A -85,B 0,C 180,E1 -7295.959,E2 -7295.959} C_VEL
LIN {X 0,Y 474.05,Z 390.87,A -85,B 0,C 180,E1 -7297.455,E2 -7297.455} C_VEL
LIN {X 0,Y 474.378,Z 384.228,A -85,B 0,C 180,E1 -7298.736,E2 -7298.736} C_VEL
LIN {X 0,Y 474.752,Z 375.984,A -85,B 0,C 180,E1 -7300.018,E2 -7300.018} C_VEL
LIN {X 0,Y 475.117,Z 367.529,A -85,B 0,C 180,E1 -7301.088,E2 -7301.088} C_VEL
LIN {X 0,Y 475.609,Z 357.095,A -85,B 0,C 180,E1 -7302.155,E2 -7302.155} C_VEL
LIN {X 0,Y 476.031,Z 346.024,A -85,B 0,C 180,E1 -7303.067,E2 -7303.067} C_VEL
LIN {X 0,Y 476.437,Z 335.384,A -85,B 0,C 180,E1 -7303.762,E2 -7303.762} C_VEL
LIN {X 0,Y 476.9,Z 323.735,A -85,B 0,C 180,E1 -7304.346,E2 -7304.346} C_VEL
LIN {X 0,Y 476.913,Z 315.412,A -85,B 0,C 180,E1 -7304.673,E2 -7304.673} C_VEL
LIN {X 0,Y 474.896,Z 302.971,A -85,B 0,C 180,E1 -7305.089,E2 -7305.089} C_VEL
LIN {X 0,Y 474.27,Z 299.453,A -85,B 0,C 180,E1 -7305.196,E2 -7305.196} C_VEL
LIN {X 0,Y 474.547,Z 288.984,A -85,B 0,C 180,E1 -7308.587,E2 -7308.587} C_VEL
LIN {X 0,Y 474.803,Z 279.424,A -85,B 0,C 180,E1 -7311.72,E2 -7311.72} C_VEL
LIN {X 0,Y 475.08,Z 269.862,A -85,B 0,C 180,E1 -7314.937,E2 -7314.937} C_VEL
LIN {X 0,Y 475.427,Z 261.618,A -85,B 0,C 180,E1 -7317.822,E2 -7317.822} C_VEL
LIN {X 0,Y 475.788,Z 252.402,A -85,B 0,C 180,E1 -7321.132,E2 -7321.132} C_VEL
LIN {X 0,Y 476.192,Z 243.988,A -85,B 0,C 180,E1 -7324.26,E2 -7324.26} C_VEL
LIN {X 0,Y 476.271,Z 239.034,A -85,B 0,C 180,E1 -7326.176,E2 -7326.176} C_VEL
LIN {X 0,Y 475.18,Z 232.401,A -85,B 0,C 180,E1 -7328.946,E2 -7328.946} C_VEL
LIN {X 0,Y 474.619,Z 229.367,A -85,B 0,C 180,E1 -7330.33,E2 -7330.33} C_VEL
LIN {X 0,Y 474.608,Z 229.368,A -85,B 0,C 180,E1 -7333.482,E2 -7333.482} C_VEL
LIN {X 0,Y 474.609,Z 229.366,A -85,B 0,C 180,E1 -7336.519,E2 -7336.519} C_VEL
LIN {X 0,Y 474.624,Z 229.367,A -85,B 0,C 180,E1 -7339.343,E2 -7339.343} C_VEL
LIN {X 0,Y 474.59,Z 229.37,A -85,B 0,C 180,E1 -7342.616,E2 -7342.616} C_VEL
LIN {X 0,Y 474.624,Z 229.36,A -85,B 0,C 180,E1 -7345.758,E2 -7345.758} C_VEL
LIN {X 0,Y 474.598,Z 229.366,A -85,B 0,C 180,E1 -7348.782,E2 -7348.782} C_VEL
LIN {X 0,Y 474.626,Z 229.364,A -85,B 0,C 180,E1 -7351.716,E2 -7351.716} C_VEL
LIN {X 0,Y 474.658,Z 229.359,A -85,B 0,C 180,E1 -7354.583,E2 -7354.583} C_VEL
LIN {X 0,Y 474.607,Z 229.366,A -85,B 0,C 180,E1 -7357.356,E2 -7357.356} C_VEL
LIN {X 0,Y 474.658,Z 229.36,A -85,B 0,C 180,E1 -7360.09,E2 -7360.09} C_VEL
LIN {X 0,Y 474.602,Z 229.366,A -85,B 0,C 180,E1 -7362.773,E2 -7362.773} C_VEL
LIN {X 0,Y 474.634,Z 229.36,A -85,B 0,C 180,E1 -7365.421,E2 -7365.421} C_VEL
LIN {X 0,Y 474.699,Z 229.355,A -85,B 0,C 180,E1 -7368.037,E2 -7368.037} C_VEL
LIN {X 0,Y 474.709,Z 229.356,A -85,B 0,C 180,E1 -7371.486,E2 -7371.486} C_VEL
LIN {X 0,Y 474.776,Z 229.344,A -85,B 0,C 180,E1 -7374.052,E2 -7374.052} C_VEL
LIN {X 0,Y 474.9,Z 229.329,A -85,B 0,C 180,E1 -7377.456,E2 -7377.456} C_VEL
LIN {X 0,Y 474.917,Z 229.329,A -85,B 0,C 180,E1 -7380,E2 -7380} C_VEL
LIN {X 0,Y 474.89,Z 229.33,A -85,B 0,C 180,E1 -7382.545,E2 -7382.545} C_VEL
LIN {X 0,Y 474.734,Z 229.348,A -85,B 0,C 180,E1 -7385.948,E2 -7385.948} C_VEL
LIN {X 0,Y 474.702,Z 229.352,A -85,B 0,C 180,E1 -7388.514,E2 -7388.514} C_VEL
LIN {X 0,Y 474.711,Z 229.352,A -85,B 0,C 180,E1 -7391.962,E2 -7391.962} C_VEL
LIN {X 0,Y 474.708,Z 229.353,A -85,B 0,C 180,E1 -7395.456,E2 -7395.456} C_VEL
LIN {X 0,Y 474.671,Z 229.358,A -85,B 0,C 180,E1 -7399.01,E2 -7399.01} C_VEL
LIN {X 0,Y 474.595,Z 229.367,A -85,B 0,C 180,E1 -7401.729,E2 -7401.729} C_VEL
LIN {X 0,Y 474.626,Z 229.363,A -85,B 0,C 180,E1 -7404.495,E2 -7404.495} C_VEL
LIN {X 0,Y 474.6,Z 229.364,A -85,B 0,C 180,E1 -7407.326,E2 -7407.326} C_VEL
LIN {X 0,Y 474.604,Z 229.367,A -85,B 0,C 180,E1 -7410.231,E2 -7410.231} C_VEL
LIN {X 0,Y 474.632,Z 229.362,A -85,B 0,C 180,E1 -7413.221,E2 -7413.221} C_VEL
LIN {X 0,Y 474.591,Z 229.368,A -85,B 0,C 180,E1 -7416.324,E2 -7416.324} C_VEL
LIN {X 0,Y 474.632,Z 229.363,A -85,B 0,C 180,E1 -7419.547,E2 -7419.547} C_VEL
LIN {X 0,Y 474.607,Z 229.366,A -85,B 0,C 180,E1 -7422.233,E2 -7422.233} C_VEL
LIN {X 0,Y 474.62,Z 229.362,A -85,B 0,C 180,E1 -7425.298,E2 -7425.298} C_VEL
LIN {X 0,Y 474.587,Z 229.37,A -85,B 0,C 180,E1 -7428.21,E2 -7428.21} C_VEL
LIN {X 0,Y 474.612,Z 229.366,A -85,B 0,C 180,E1 -7431.541,E2 -7431.541} C_VEL
LIN {X 0,Y 474.628,Z 229.364,A -85,B 0,C 180,E1 -7434.725,E2 -7434.725} C_VEL
LIN {X 0,Y 474.609,Z 229.365,A -85,B 0,C 180,E1 -7437.784,E2 -7437.784} C_VEL
LIN {X 0,Y 474.296,Z 229.407,A -85,B 0,C 180,E1 -7440.957,E2 -7440.957} C_VEL
LIN {X 0,Y 474.165,Z 229.425,A -85,B 0,C 180,E1 -7441.685,E2 -7441.685} C_VEL
LIN {X 0,Y 474.136,Z 232.437,A -85,B 0,C 180,E1 -7444.715,E2 -7444.715} C_VEL
LIN {X 0,Y 474.051,Z 235.168,A -85,B 0,C 180,E1 -7447.326,E2 -7447.326} C_VEL
LIN {X 0,Y 474.007,Z 238.055,A -85,B 0,C 180,E1 -7450.06,E2 -7450.06} C_VEL
LIN {X 0,Y 474.01,Z 239.604,A -85,B 0,C 180,E1 -7451.508,E2 -7451.508} C_VEL
LIN {X 0,Y 473.387,Z 240.419,A -85,B 0,C 180,E1 -7452.21,E2 -7452.21} C_VEL
LIN {X 0,Y 470.562,Z 241.933,A -85,B 0,C 180,E1 -7453.347,E2 -7453.347} C_VEL
LIN {X 0,Y 468.122,Z 243.174,A -85,B 0,C 180,E1 -7454.263,E2 -7454.263} C_VEL
LIN {X 0,Y 467.038,Z 244.059,A -85,B 0,C 180,E1 -7454.972,E2 -7454.972} C_VEL
LIN {X 0,Y 466.931,Z 244.335,A -85,B 0,C 180,E1 -7455.212,E2 -7455.212} C_VEL
LIN {X 0,Y 466.92,Z 248.364,A -85,B 0,C 180,E1 -7458.742,E2 -7458.742} C_VEL
LIN {X 0,Y 470.18,Z 262.651,A -85,B 0,C 180,E1 -7459.285,E2 -7459.285} C_VEL
LIN {X 0,Y 470.09,Z 274.744,A -85,B 0,C 180,E1 -7459.827,E2 -7459.827} C_VEL
LIN {X 0,Y 469.684,Z 286.439,A -85,B 0,C 180,E1 -7460.525,E2 -7460.525} C_VEL
LIN {X 0,Y 469.102,Z 297.7,A -85,B 0,C 180,E1 -7461.382,E2 -7461.382} C_VEL
LIN {X 0,Y 468.763,Z 307.827,A -85,B 0,C 180,E1 -7462.352,E2 -7462.352} C_VEL
LIN {X 0,Y 468.33,Z 316.132,A -85,B 0,C 180,E1 -7463.32,E2 -7463.32} C_VEL
LIN {X 0,Y 467.849,Z 325.135,A -85,B 0,C 180,E1 -7464.612,E2 -7464.612} C_VEL
LIN {X 0,Y 467.484,Z 332.388,A -85,B 0,C 180,E1 -7465.904,E2 -7465.904} C_VEL
LIN {X 0,Y 466.965,Z 339.079,A -85,B 0,C 180,E1 -7467.411,E2 -7467.411} C_VEL
LIN {X 0,Y 466.936,Z 343.472,A -85,B 0,C 180,E1 -7468.705,E2 -7468.705} C_VEL
LIN {X 0,Y 466.689,Z 346.834,A -85,B 0,C 180,E1 -7469.999,E2 -7469.999} C_VEL
LIN {X 0,Y 466.706,Z 349.763,A -85,B 0,C 180,E1 -7471.725,E2 -7471.725} C_VEL
LIN {X 0,Y 466.803,Z 350.642,A -85,B 0,C 180,E1 -7472.587,E2 -7472.587} C_VEL
LIN {X 0,Y 466.798,Z 351.119,A -85,B 0,C 180,E1 -7473.451,E2 -7473.451} C_VEL
LIN {X 0,Y 466.717,Z 350.885,A -85,B 0,C 180,E1 -7475.182,E2 -7475.182} C_VEL
LIN {X 0,Y 466.8,Z 349.728,A -85,B 0,C 180,E1 -7476.443,E2 -7476.443} C_VEL
LIN {X 0,Y 466.848,Z 347.561,A -85,B 0,C 180,E1 -7477.785,E2 -7477.785} C_VEL
LIN {X 0,Y 466.952,Z 344.471,A -85,B 0,C 180,E1 -7479.091,E2 -7479.091} C_VEL
LIN {X 0,Y 467.082,Z 340.319,A -85,B 0,C 180,E1 -7480.401,E2 -7480.401} C_VEL
LIN {X 0,Y 467.414,Z 333.97,A -85,B 0,C 180,E1 -7481.93,E2 -7481.93} C_VEL
LIN {X 0,Y 467.794,Z 327.012,A -85,B 0,C 180,E1 -7483.243,E2 -7483.243} C_VEL
LIN {X 0,Y 468.246,Z 318.258,A -85,B 0,C 180,E1 -7484.559,E2 -7484.559} C_VEL
LIN {X 0,Y 468.713,Z 309.259,A -85,B 0,C 180,E1 -7485.657,E2 -7485.657} C_VEL
LIN {X 0,Y 469.184,Z 299.314,A -85,B 0,C 180,E1 -7486.646,E2 -7486.646} C_VEL
LIN {X 0,Y 469.687,Z 288.209,A -85,B 0,C 180,E1 -7487.524,E2 -7487.524} C_VEL
LIN {X 0,Y 470.142,Z 275.715,A -85,B 0,C 180,E1 -7488.294,E2 -7488.294} C_VEL
LIN {X 0,Y 470.382,Z 262.94,A -85,B 0,C 180,E1 -7488.877,E2 -7488.877} C_VEL
LIN {X 0,Y 467.236,Z 250.148,A -85,B 0,C 180,E1 -7489.394,E2 -7489.394} C_VEL
LIN {X 0,Y 466.87,Z 248.451,A -85,B 0,C 180,E1 -7489.453,E2 -7489.453} C_VEL
LIN {X 0,Y 466.891,Z 244.465,A -85,B 0,C 180,E1 -7493.038,E2 -7493.038} C_VEL
LIN {X 0,Y 466.976,Z 241.386,A -85,B 0,C 180,E1 -7495.876,E2 -7495.876} C_VEL
LIN {X 0,Y 467.045,Z 237.918,A -85,B 0,C 180,E1 -7499.217,E2 -7499.217} C_VEL
LIN {X 0,Y 467.115,Z 234.475,A -85,B 0,C 180,E1 -7502.589,E2 -7502.589} C_VEL
LIN {X 0,Y 467.179,Z 231.395,A -85,B 0,C 180,E1 -7505.673,E2 -7505.673} C_VEL
LIN {X 0,Y 467.247,Z 230.287,A -85,B 0,C 180,E1 -7507.137,E2 -7507.137} C_VEL
LIN {X 0,Y 467.529,Z 230.246,A -85,B 0,C 180,E1 -7509.946,E2 -7509.946} C_VEL
LIN {X 0,Y 467.58,Z 230.244,A -85,B 0,C 180,E1 -7512.566,E2 -7512.566} C_VEL
LIN {X 0,Y 467.563,Z 230.242,A -85,B 0,C 180,E1 -7515.052,E2 -7515.052} C_VEL
LIN {X 0,Y 467.565,Z 230.242,A -85,B 0,C 180,E1 -7518.595,E2 -7518.595} C_VEL
LIN {X 0,Y 467.558,Z 230.243,A -85,B 0,C 180,E1 -7521.954,E2 -7521.954} C_VEL
LIN {X 0,Y 467.558,Z 230.243,A -85,B 0,C 180,E1 -7525.167,E2 -7525.167} C_VEL
LIN {X 0,Y 467.572,Z 230.24,A -85,B 0,C 180,E1 -7528.259,E2 -7528.259} C_VEL
LIN {X 0,Y 467.567,Z 230.242,A -85,B 0,C 180,E1 -7531.25,E2 -7531.25} C_VEL
LIN {X 0,Y 467.602,Z 230.242,A -85,B 0,C 180,E1 -7534.159,E2 -7534.159} C_VEL
LIN {X 0,Y 467.567,Z 230.243,A -85,B 0,C 180,E1 -7536.995,E2 -7536.995} C_VEL
LIN {X 0,Y 467.611,Z 230.235,A -85,B 0,C 180,E1 -7539.776,E2 -7539.776} C_VEL
LIN {X 0,Y 467.596,Z 230.242,A -85,B 0,C 180,E1 -7542.506,E2 -7542.506} C_VEL
LIN {X 0,Y 467.595,Z 230.239,A -85,B 0,C 180,E1 -7545.196,E2 -7545.196} C_VEL
LIN {X 0,Y 467.644,Z 230.232,A -85,B 0,C 180,E1 -7547.854,E2 -7547.854} C_VEL
LIN {X 0,Y 467.667,Z 230.229,A -85,B 0,C 180,E1 -7551.357,E2 -7551.357} C_VEL
LIN {X 0,Y 467.744,Z 230.224,A -85,B 0,C 180,E1 -7553.962,E2 -7553.962} C_VEL
LIN {X 0,Y 467.849,Z 230.209,A -85,B 0,C 180,E1 -7557.417,E2 -7557.417} C_VEL
LIN {X 0,Y 467.866,Z 230.205,A -85,B 0,C 180,E1 -7560,E2 -7560} C_VEL
LIN {X 0,Y 467.849,Z 230.207,A -85,B 0,C 180,E1 -7562.583,E2 -7562.583} C_VEL
LIN {X 0,Y 467.742,Z 230.22,A -85,B 0,C 180,E1 -7566.037,E2 -7566.037} C_VEL
LIN {X 0,Y 467.669,Z 230.233,A -85,B 0,C 180,E1 -7568.643,E2 -7568.643} C_VEL
LIN {X 0,Y 467.644,Z 230.235,A -85,B 0,C 180,E1 -7572.146,E2 -7572.146} C_VEL
LIN {X 0,Y 467.628,Z 230.233,A -85,B 0,C 180,E1 -7575.695,E2 -7575.695} C_VEL
LIN {X 0,Y 467.606,Z 230.238,A -85,B 0,C 180,E1 -7578.765,E2 -7578.765} C_VEL
LIN {X 0,Y 467.569,Z 230.241,A -85,B 0,C 180,E1 -7581.269,E2 -7581.269} C_VEL
LIN {X 0,Y 467.558,Z 230.244,A -85,B 0,C 180,E1 -7583.944,E2 -7583.944} C_VEL
LIN {X 0,Y 467.617,Z 230.24,A -85,B 0,C 180,E1 -7586.8,E2 -7586.8} C_VEL
LIN {X 0,Y 467.577,Z 230.242,A -85,B 0,C 180,E1 -7589.737,E2 -7589.737} C_VEL
LIN {X 0,Y 467.573,Z 230.241,A -85,B 0,C 180,E1 -7592.759,E2 -7592.759} C_VEL
LIN {X 0,Y 467.544,Z 230.245,A -85,B 0,C 180,E1 -7595.891,E2 -7595.891} C_VEL
LIN {X 0,Y 467.574,Z 230.241,A -85,B 0,C 180,E1 -7599.146,E2 -7599.146} C_VEL
LIN {X 0,Y 467.567,Z 230.244,A -85,B 0,C 180,E1 -7601.404,E2 -7601.404} C_VEL
LIN {X 0,Y 467.562,Z 230.246,A -85,B 0,C 180,E1 -7605.054,E2 -7605.054} C_VEL
LIN {X 0,Y 467.582,Z 230.243,A -85,B 0,C 180,E1 -7607.441,E2 -7607.441} C_VEL
LIN {X 0,Y 467.595,Z 230.257,A -85,B 0,C 180,E1 -7609.173,E2 -7609.173} C_VEL
LIN {X 0,Y 468.73,Z 236.559,A -85,B 0,C 180,E1 -7612.069,E2 -7612.069} C_VEL
LIN {X 0,Y 469.325,Z 240.958,A -85,B 0,C 180,E1 -7613.963,E2 -7613.963} C_VEL
LIN {X 0,Y 469.127,Z 246.918,A -85,B 0,C 180,E1 -7616.339,E2 -7616.339} C_VEL
LIN {X 0,Y 468.739,Z 254.844,A -85,B 0,C 180,E1 -7619.353,E2 -7619.353} C_VEL
LIN {X 0,Y 468.33,Z 264.234,A -85,B 0,C 180,E1 -7622.763,E2 -7622.763} C_VEL
LIN {X 0,Y 467.906,Z 273.651,A -85,B 0,C 180,E1 -7626.076,E2 -7626.076} C_VEL
LIN {X 0,Y 467.623,Z 283.229,A -85,B 0,C 180,E1 -7629.319,E2 -7629.319} C_VEL
LIN {X 0,Y 467.394,Z 291.47,A -85,B 0,C 180,E1 -7632.048,E2 -7632.048} C_VEL
LIN {X 0,Y 467.229,Z 299.134,A -85,B 0,C 180,E1 -7634.572,E2 -7634.572} C_VEL
LIN {X 0,Y 469.828,Z 314.76,A -85,B 0,C 180,E1 -7635.089,E2 -7635.089} C_VEL
LIN {X 0,Y 470.103,Z 319.596,A -85,B 0,C 180,E1 -7635.278,E2 -7635.278} C_VEL
